LIN {X 0,Y 267.392,Z 674.93,A -85,B 0,C 180,E1 -18340.221,E2 -18340.221} C_VEL
LIN {X 0,Y 266.458,Z 688.326,A -85,B 0,C 180,E1 -18341.349,E2 -18341.349} C_VEL
LIN {X 0,Y 265.506,Z 700.294,A -85,B 0,C 180,E1 -18342.659,E2 -18342.659} C_VEL
LIN {X 0,Y 264.466,Z 712.728,A -85,B 0,C 180,E1 -18344.391,E2 -18344.391} C_VEL
LIN {X 0,Y 263.562,Z 722.705,A -85,B 0,C 180,E1 -18346.114,E2 -18346.114} C_VEL
LIN {X 0,Y 263.255,Z 725.943,A -85,B 0,C 180,E1 -18346.753,E2 -18346.753} C_VEL
LIN {X 0,Y 262.224,Z 730.137,A -85,B 0,C 180,E1 -18347.633,E2 -18347.633} C_VEL
LIN {X 0,Y 258.805,Z 736.401,A -85,B 0,C 180,E1 -18349.151,E2 -18349.151} C_VEL
LIN {X 0,Y 255.472,Z 742.099,A -85,B 0,C 180,E1 -18350.814,E2 -18350.814} C_VEL
LIN {X 0,Y 254.593,Z 745.41,A -85,B 0,C 180,E1 -18351.903,E2 -18351.903} C_VEL
LIN {X 0,Y 254.229,Z 751.934,A -85,B 0,C 180,E1 -18354.384,E2 -18354.384} C_VEL
LIN {X 0,Y 254.116,Z 756.958,A -85,B 0,C 180,E1 -18356.829,E2 -18356.829} C_VEL
LIN {X 0,Y 254.037,Z 760.636,A -85,B 0,C 180,E1 -18359.207,E2 -18359.207} C_VEL
LIN {X 0,Y 254.108,Z 763.255,A -85,B 0,C 180,E1 -18361.585,E2 -18361.585} C_VEL
LIN {X 0,Y 254.189,Z 764.422,A -85,B 0,C 180,E1 -18363.17,E2 -18363.17} C_VEL
LIN {X 0,Y 254.813,Z 765.536,A -85,B 0,C 180,E1 -18366.334,E2 -18366.334} C_VEL
LIN {X 0,Y 255.358,Z 765.437,A -85,B 0,C 180,E1 -18367.91,E2 -18367.91} C_VEL
LIN {X 0,Y 255.895,Z 764.932,A -85,B 0,C 180,E1 -18369.485,E2 -18369.485} C_VEL
LIN {X 0,Y 257.702,Z 762.72,A -85,B 0,C 180,E1 -18372.602,E2 -18372.602} C_VEL
LIN {X 0,Y 259.373,Z 759.949,A -85,B 0,C 180,E1 -18374.917,E2 -18374.917} C_VEL
LIN {X 0,Y 261.617,Z 756.12,A -85,B 0,C 180,E1 -18377.188,E2 -18377.188} C_VEL
LIN {X 0,Y 264.305,Z 751.227,A -85,B 0,C 180,E1 -18379.413,E2 -18379.413} C_VEL
LIN {X 0,Y 267.393,Z 745.066,A -85,B 0,C 180,E1 -18381.59,E2 -18381.59} C_VEL
LIN {X 0,Y 271.525,Z 736.165,A -85,B 0,C 180,E1 -18384.058,E2 -18384.058} C_VEL
LIN {X 0,Y 275.529,Z 726.618,A -85,B 0,C 180,E1 -18386.098,E2 -18386.098} C_VEL
LIN {X 0,Y 279.335,Z 716.352,A -85,B 0,C 180,E1 -18387.872,E2 -18387.872} C_VEL
LIN {X 0,Y 282.742,Z 706.311,A -85,B 0,C 180,E1 -18389.245,E2 -18389.245} C_VEL
LIN {X 0,Y 286.702,Z 692.836,A -85,B 0,C 180,E1 -18390.701,E2 -18390.701} C_VEL
LIN {X 0,Y 290.054,Z 679.318,A -85,B 0,C 180,E1 -18391.803,E2 -18391.803} C_VEL
LIN {X 0,Y 292.766,Z 665.226,A -85,B 0,C 180,E1 -18392.641,E2 -18392.641} C_VEL
LIN {X 0,Y 303.886,Z 598.397,A -85,B 0,C 180,E1 -18395.644,E2 -18395.644} C_VEL
LIN {X 0,Y 304.018,Z 586.794,A -85,B 0,C 180,E1 -18397.144,E2 -18397.144} C_VEL
LIN {X 0,Y 303.238,Z 583.136,A -85,B 0,C 180,E1 -18398.173,E2 -18398.173} C_VEL
LIN {X 0,Y 302.067,Z 579.008,A -85,B 0,C 180,E1 -18399.844,E2 -18399.844} C_VEL
LIN {X 0,Y 301.134,Z 575.43,A -85,B 0,C 180,E1 -18401.899,E2 -18401.899} C_VEL
LIN {X 0,Y 300.72,Z 573.5,A -85,B 0,C 180,E1 -18404.044,E2 -18404.044} C_VEL
LIN {X 0,Y 301.094,Z 572.833,A -85,B 0,C 180,E1 -18406.352,E2 -18406.352} C_VEL
LIN {X 0,Y 302.26,Z 573.558,A -85,B 0,C 180,E1 -18408.617,E2 -18408.617} C_VEL
LIN {X 0,Y 304.282,Z 575.713,A -85,B 0,C 180,E1 -18410.892,E2 -18410.892} C_VEL
LIN {X 0,Y 305.244,Z 577.018,A -85,B 0,C 180,E1 -18411.75,E2 -18411.75} C_VEL
LIN {X 0,Y 305.469,Z 578.807,A -85,B 0,C 180,E1 -18412.164,E2 -18412.164} C_VEL
LIN {X 0,Y 290.536,Z 664.644,A -85,B 0,C 180,E1 -18416.195,E2 -18416.195} C_VEL
LIN {X 0,Y 287.406,Z 682.317,A -85,B 0,C 180,E1 -18417.142,E2 -18417.142} C_VEL
LIN {X 0,Y 284.436,Z 695.44,A -85,B 0,C 180,E1 -18418.12,E2 -18418.12} C_VEL
LIN {X 0,Y 280.955,Z 708.177,A -85,B 0,C 180,E1 -18419.358,E2 -18419.358} C_VEL
LIN {X 0,Y 277.428,Z 719.855,A -85,B 0,C 180,E1 -18420.813,E2 -18420.813} C_VEL
LIN {X 0,Y 273.027,Z 732.546,A -85,B 0,C 180,E1 -18422.812,E2 -18422.812} C_VEL
LIN {X 0,Y 269.061,Z 742.824,A -85,B 0,C 180,E1 -18424.884,E2 -18424.884} C_VEL
LIN {X 0,Y 265.679,Z 751.358,A -85,B 0,C 180,E1 -18427.034,E2 -18427.034} C_VEL
LIN {X 0,Y 262.22,Z 759.42,A -85,B 0,C 180,E1 -18429.609,E2 -18429.609} C_VEL
LIN {X 0,Y 259.817,Z 765.006,A -85,B 0,C 180,E1 -18431.876,E2 -18431.876} C_VEL
LIN {X 0,Y 257.299,Z 770.761,A -85,B 0,C 180,E1 -18434.96,E2 -18434.96} C_VEL
LIN {X 0,Y 255.921,Z 773.892,A -85,B 0,C 180,E1 -18437.309,E2 -18437.309} C_VEL
LIN {X 0,Y 254.674,Z 776.576,A -85,B 0,C 180,E1 -18440.469,E2 -18440.469} C_VEL
LIN {X 0,Y 254.325,Z 777.326,A -85,B 0,C 180,E1 -18442.058,E2 -18442.058} C_VEL
LIN {X 0,Y 254.021,Z 777.636,A -85,B 0,C 180,E1 -18444.881,E2 -18444.881} C_VEL
LIN {X 0,Y 254.106,Z 777.04,A -85,B 0,C 180,E1 -18446.829,E2 -18446.829} C_VEL
LIN {X 0,Y 254.099,Z 775.415,A -85,B 0,C 180,E1 -18449.307,E2 -18449.307} C_VEL
LIN {X 0,Y 254.062,Z 777.171,A -85,B 0,C 180,E1 -18451.585,E2 -18451.585} C_VEL
LIN {X 0,Y 254.068,Z 777.92,A -85,B 0,C 180,E1 -18453.172,E2 -18453.172} C_VEL
LIN {X 0,Y 254.058,Z 778.293,A -85,B 0,C 180,E1 -18456.353,E2 -18456.353} C_VEL
LIN {X 0,Y 254.583,Z 777.255,A -85,B 0,C 180,E1 -18459.534,E2 -18459.534} C_VEL
LIN {X 0,Y 255.697,Z 774.838,A -85,B 0,C 180,E1 -18462.702,E2 -18462.702} C_VEL
LIN {X 0,Y 257.682,Z 771.008,A -85,B 0,C 180,E1 -18465.828,E2 -18465.828} C_VEL
LIN {X 0,Y 260.158,Z 765.718,A -85,B 0,C 180,E1 -18468.916,E2 -18468.916} C_VEL
LIN {X 0,Y 262.696,Z 760.659,A -85,B 0,C 180,E1 -18471.172,E2 -18471.172} C_VEL
LIN {X 0,Y 266.135,Z 753.523,A -85,B 0,C 180,E1 -18473.748,E2 -18473.748} C_VEL
LIN {X 0,Y 270.246,Z 744.85,A -85,B 0,C 180,E1 -18476.238,E2 -18476.238} C_VEL
LIN {X 0,Y 274.277,Z 735.941,A -85,B 0,C 180,E1 -18478.297,E2 -18478.297} C_VEL
LIN {X 0,Y 278.781,Z 725.251,A -85,B 0,C 180,E1 -18480.278,E2 -18480.278} C_VEL
LIN {X 0,Y 283.286,Z 713.812,A -85,B 0,C 180,E1 -18481.991,E2 -18481.991} C_VEL
LIN {X 0,Y 287.778,Z 700.836,A -85,B 0,C 180,E1 -18483.546,E2 -18483.546} C_VEL
LIN {X 0,Y 291.653,Z 688.544,A -85,B 0,C 180,E1 -18484.701,E2 -18484.701} C_VEL
LIN {X 0,Y 295.512,Z 674.017,A -85,B 0,C 180,E1 -18485.744,E2 -18485.744} C_VEL
LIN {X 0,Y 298.806,Z 658.507,A -85,B 0,C 180,E1 -18486.571,E2 -18486.571} C_VEL
LIN {X 0,Y 310.853,Z 589.993,A -85,B 0,C 180,E1 -18489.42,E2 -18489.42} C_VEL
LIN {X 0,Y 309.732,Z 587.337,A -85,B 0,C 180,E1 -18490.47,E2 -18490.47} C_VEL
LIN {X 0,Y 308.475,Z 584.65,A -85,B 0,C 180,E1 -18491.851,E2 -18491.851} C_VEL
LIN {X 0,Y 307.029,Z 581.664,A -85,B 0,C 180,E1 -18494.357,E2 -18494.357} C_VEL
LIN {X 0,Y 306.336,Z 581.501,A -85,B 0,C 180,E1 -18497.236,E2 -18497.236} C_VEL
LIN {X 0,Y 306.709,Z 582.69,A -85,B 0,C 180,E1 -18499.243,E2 -18499.243} C_VEL
LIN {X 0,Y 308.011,Z 587.255,A -85,B 0,C 180,E1 -18502.044,E2 -18502.044} C_VEL
LIN {X 0,Y 309.168,Z 591.574,A -85,B 0,C 180,E1 -18503.631,E2 -18503.631} C_VEL
LIN {X 0,Y 309.454,Z 593.023,A -85,B 0,C 180,E1 -18504.035,E2 -18504.035} C_VEL
LIN {X 0,Y 309.128,Z 598.033,A -85,B 0,C 180,E1 -18504.592,E2 -18504.592} C_VEL
LIN {X 0,Y 297.304,Z 660.919,A -85,B 0,C 180,E1 -18507.467,E2 -18507.467} C_VEL
LIN {X 0,Y 294.179,Z 674.017,A -85,B 0,C 180,E1 -18508.292,E2 -18508.292} C_VEL
LIN {X 0,Y 290.356,Z 687.818,A -85,B 0,C 180,E1 -18509.449,E2 -18509.449} C_VEL
LIN {X 0,Y 286.275,Z 700.375,A -85,B 0,C 180,E1 -18510.795,E2 -18510.795} C_VEL
LIN {X 0,Y 281.68,Z 712.899,A -85,B 0,C 180,E1 -18512.511,E2 -18512.511} C_VEL
LIN {X 0,Y 277.789,Z 722.415,A -85,B 0,C 180,E1 -18514.124,E2 -18514.124} C_VEL
LIN {X 0,Y 272.883,Z 733.435,A -85,B 0,C 180,E1 -18516.472,E2 -18516.472} C_VEL
LIN {X 0,Y 269.093,Z 741.153,A -85,B 0,C 180,E1 -18518.553,E2 -18518.553} C_VEL
LIN {X 0,Y 265.844,Z 747.53,A -85,B 0,C 180,E1 -18520.703,E2 -18520.703} C_VEL
LIN {X 0,Y 263.047,Z 752.715,A -85,B 0,C 180,E1 -18522.909,E2 -18522.909} C_VEL
LIN {X 0,Y 259.802,Z 758.061,A -85,B 0,C 180,E1 -18525.909,E2 -18525.909} C_VEL
LIN {X 0,Y 258.501,Z 760.04,A -85,B 0,C 180,E1 -18527.438,E2 -18527.438} C_VEL
LIN {X 0,Y 256.764,Z 762.528,A -85,B 0,C 180,E1 -18530.19,E2 -18530.19} C_VEL
LIN {X 0,Y 255.749,Z 763.559,A -85,B 0,C 180,E1 -18532.103,E2 -18532.103} C_VEL
LIN {X 0,Y 255.112,Z 763.932,A -85,B 0,C 180,E1 -18533.673,E2 -18533.673} C_VEL
LIN {X 0,Y 254.722,Z 763.876,A -85,B 0,C 180,E1 -18535.252,E2 -18535.252} C_VEL
LIN {X 0,Y 254.423,Z 763.427,A -85,B 0,C 180,E1 -18536.833,E2 -18536.833} C_VEL
LIN {X 0,Y 254.191,Z 762.579,A -85,B 0,C 180,E1 -18538.416,E2 -18538.416} C_VEL
LIN {X 0,Y 254.082,Z 761.32,A -85,B 0,C 180,E1 -18540,E2 -18540} C_VEL
LIN {X 0,Y 254.026,Z 758.577,A -85,B 0,C 180,E1 -18542.378,E2 -18542.378} C_VEL
LIN {X 0,Y 254.063,Z 754.795,A -85,B 0,C 180,E1 -18544.76,E2 -18544.76} C_VEL
LIN {X 0,Y 254.334,Z 749.877,A -85,B 0,C 180,E1 -18547.143,E2 -18547.143} C_VEL
LIN {X 0,Y 254.694,Z 743.632,A -85,B 0,C 180,E1 -18549.53,E2 -18549.53} C_VEL
LIN {X 0,Y 255.279,Z 735.844,A -85,B 0,C 180,E1 -18551.916,E2 -18551.916} C_VEL
LIN {X 0,Y 256.201,Z 726.268,A -85,B 0,C 180,E1 -18554.293,E2 -18554.293} C_VEL
LIN {X 0,Y 256.973,Z 716.914,A -85,B 0,C 180,E1 -18556.203,E2 -18556.203} C_VEL
LIN {X 0,Y 258.209,Z 705.975,A -85,B 0,C 180,E1 -18558.036,E2 -18558.036} C_VEL
LIN {X 0,Y 259.48,Z 693.061,A -85,B 0,C 180,E1 -18559.789,E2 -18559.789} C_VEL
LIN {X 0,Y 260.62,Z 679.32,A -85,B 0,C 180,E1 -18561.245,E2 -18561.245} C_VEL
LIN {X 0,Y 261.707,Z 665.038,A -85,B 0,C 180,E1 -18562.396,E2 -18562.396} C_VEL
LIN {X 0,Y 262.599,Z 649.769,A -85,B 0,C 180,E1 -18563.251,E2 -18563.251} C_VEL
LIN {X 0,Y 266.046,Z 579.424,A -85,B 0,C 180,E1 -18566.286,E2 -18566.286} C_VEL
LIN {X 0,Y 262.645,Z 547.859,A -85,B 0,C 180,E1 -18567.923,E2 -18567.923} C_VEL
LIN {X 0,Y 261.965,Z 538.359,A -85,B 0,C 180,E1 -18568.424,E2 -18568.424} C_VEL
LIN {X 0,Y 262.567,Z 533.905,A -85,B 0,C 180,E1 -18569.682,E2 -18569.682} C_VEL
LIN {X 0,Y 260.638,Z 524.372,A -85,B 0,C 180,E1 -18572.635,E2 -18572.635} C_VEL
LIN {X 0,Y 258.14,Z 512.652,A -85,B 0,C 180,E1 -18576.425,E2 -18576.425} C_VEL
LIN {X 0,Y 256.098,Z 503.706,A -85,B 0,C 180,E1 -18579.458,E2 -18579.458} C_VEL
LIN {X 0,Y 256.065,Z 503.713,A -85,B 0,C 180,E1 -18583.326,E2 -18583.326} C_VEL
LIN {X 0,Y 256.073,Z 503.714,A -85,B 0,C 180,E1 -18587.819,E2 -18587.819} C_VEL
LIN {X 0,Y 256.073,Z 503.711,A -85,B 0,C 180,E1 -18590.858,E2 -18590.858} C_VEL
LIN {X 0,Y 256.11,Z 503.704,A -85,B 0,C 180,E1 -18594.811,E2 -18594.811} C_VEL
LIN {X 0,Y 256.094,Z 503.707,A -85,B 0,C 180,E1 -18598.572,E2 -18598.572} C_VEL
LIN {X 0,Y 256.143,Z 503.701,A -85,B 0,C 180,E1 -18602.196,E2 -18602.196} C_VEL
LIN {X 0,Y 256.169,Z 503.701,A -85,B 0,C 180,E1 -18605.699,E2 -18605.699} C_VEL
LIN {X 0,Y 256.168,Z 503.7,A -85,B 0,C 180,E1 -18609.105,E2 -18609.105} C_VEL
LIN {X 0,Y 256.302,Z 503.682,A -85,B 0,C 180,E1 -18614.085,E2 -18614.085} C_VEL
LIN {X 0,Y 256.311,Z 503.681,A -85,B 0,C 180,E1 -18618.934,E2 -18618.934} C_VEL
LIN {X 0,Y 256.542,Z 503.651,A -85,B 0,C 180,E1 -18622.127,E2 -18622.127} C_VEL
LIN {X 0,Y 256.719,Z 503.628,A -85,B 0,C 180,E1 -18628.431,E2 -18628.431} C_VEL
LIN {X 0,Y 256.716,Z 503.633,A -85,B 0,C 180,E1 -18631.569,E2 -18631.569} C_VEL
LIN {X 0,Y 256.541,Z 503.651,A -85,B 0,C 180,E1 -18637.873,E2 -18637.873} C_VEL
LIN {X 0,Y 256.311,Z 503.682,A -85,B 0,C 180,E1 -18641.066,E2 -18641.066} C_VEL
LIN {X 0,Y 256.301,Z 503.681,A -85,B 0,C 180,E1 -18645.915,E2 -18645.915} C_VEL
LIN {X 0,Y 256.168,Z 503.699,A -85,B 0,C 180,E1 -18650.895,E2 -18650.895} C_VEL
LIN {X 0,Y 256.189,Z 503.697,A -85,B 0,C 180,E1 -18655.138,E2 -18655.138} C_VEL
LIN {X 0,Y 256.104,Z 503.709,A -85,B 0,C 180,E1 -18659.601,E2 -18659.601} C_VEL
LIN {X 0,Y 256.086,Z 503.711,A -85,B 0,C 180,E1 -18663.29,E2 -18663.29} C_VEL
LIN {X 0,Y 256.13,Z 503.707,A -85,B 0,C 180,E1 -18667.275,E2 -18667.275} C_VEL
LIN {X 0,Y 256.059,Z 503.715,A -85,B 0,C 180,E1 -18671.203,E2 -18671.203} C_VEL
LIN {X 0,Y 256.063,Z 503.714,A -85,B 0,C 180,E1 -18675.529,E2 -18675.529} C_VEL
LIN {X 0,Y 256.056,Z 503.713,A -85,B 0,C 180,E1 -18678.797,E2 -18678.797} C_VEL
LIN {X 0,Y 256.173,Z 503.781,A -85,B 0,C 180,E1 -18683.581,E2 -18683.581} C_VEL
LIN {X 0,Y 260.085,Z 520.834,A -85,B 0,C 180,E1 -18687.745,E2 -18687.745} C_VEL
LIN {X 0,Y 262.856,Z 533.76,A -85,B 0,C 180,E1 -18690.794,E2 -18690.794} C_VEL
LIN {X 0,Y 261.899,Z 545.387,A -85,B 0,C 180,E1 -18693.29,E2 -18693.29} C_VEL
LIN {X 0,Y 261.425,Z 550.677,A -85,B 0,C 180,E1 -18694.364,E2 -18694.364} C_VEL
LIN {X 0,Y 263.474,Z 573.72,A -85,B 0,C 180,E1 -18695.465,E2 -18695.465} C_VEL
LIN {X 0,Y 264.373,Z 582.285,A -85,B 0,C 180,E1 -18695.876,E2 -18695.876} C_VEL
LIN {X 0,Y 261.074,Z 660.539,A -85,B 0,C 180,E1 -18699.206,E2 -18699.206} C_VEL
LIN {X 0,Y 260.346,Z 674.677,A -85,B 0,C 180,E1 -18700.074,E2 -18700.074} C_VEL
LIN {X 0,Y 259.423,Z 687.6,A -85,B 0,C 180,E1 -18701.182,E2 -18701.182} C_VEL
LIN {X 0,Y 258.394,Z 700.276,A -85,B 0,C 180,E1 -18702.591,E2 -18702.591} C_VEL
LIN {X 0,Y 257.367,Z 712.658,A -85,B 0,C 180,E1 -18704.356,E2 -18704.356} C_VEL
LIN {X 0,Y 256.452,Z 722.704,A -85,B 0,C 180,E1 -18706.126,E2 -18706.126} C_VEL
LIN {X 0,Y 255.507,Z 733.568,A -85,B 0,C 180,E1 -18708.497,E2 -18708.497} C_VEL
LIN {X 0,Y 254.813,Z 742.226,A -85,B 0,C 180,E1 -18710.875,E2 -18710.875} C_VEL
LIN {X 0,Y 254.593,Z 745.41,A -85,B 0,C 180,E1 -18711.903,E2 -18711.903} C_VEL
LIN {X 0,Y 253.763,Z 748.506,A -85,B 0,C 180,E1 -18713.022,E2 -18713.022} C_VEL
LIN {X 0,Y 250.712,Z 752.886,A -85,B 0,C 180,E1 -18714.919,E2 -18714.919} C_VEL
LIN {X 0,Y 247.72,Z 756.704,A -85,B 0,C 180,E1 -18716.932,E2 -18716.932} C_VEL
LIN {X 0,Y 247.008,Z 758.795,A -85,B 0,C 180,E1 -18718.21,E2 -18718.21} C_VEL
LIN {X 0,Y 246.984,Z 761.253,A -85,B 0,C 180,E1 -18720,E2 -18720} C_VEL
LIN {X 0,Y 247.04,Z 763.011,A -85,B 0,C 180,E1 -18721.63,E2 -18721.63} C_VEL
LIN {X 0,Y 247.113,Z 764.353,A -85,B 0,C 180,E1 -18723.261,E2 -18723.261} C_VEL
LIN {X 0,Y 247.336,Z 765.232,A -85,B 0,C 180,E1 -18724.89,E2 -18724.89} C_VEL
LIN {X 0,Y 248.143,Z 765.789,A -85,B 0,C 180,E1 -18727.57,E2 -18727.57} C_VEL
LIN {X 0,Y 248.911,Z 765.442,A -85,B 0,C 180,E1 -18729.754,E2 -18729.754} C_VEL
LIN {X 0,Y 249.753,Z 764.668,A -85,B 0,C 180,E1 -18731.36,E2 -18731.36} C_VEL
LIN {X 0,Y 250.832,Z 763.486,A -85,B 0,C 180,E1 -18732.953,E2 -18732.953} C_VEL
LIN {X 0,Y 253.27,Z 759.929,A -85,B 0,C 180,E1 -18736.111,E2 -18736.111} C_VEL
LIN {X 0,Y 255.871,Z 756.046,A -85,B 0,C 180,E1 -18738.413,E2 -18738.413} C_VEL
LIN {X 0,Y 258.819,Z 751.037,A -85,B 0,C 180,E1 -18740.671,E2 -18740.671} C_VEL
LIN {X 0,Y 262.845,Z 743.72,A -85,B 0,C 180,E1 -18743.228,E2 -18743.228} C_VEL
LIN {X 0,Y 266.715,Z 735.856,A -85,B 0,C 180,E1 -18745.353,E2 -18745.353} C_VEL
LIN {X 0,Y 271.072,Z 726.284,A -85,B 0,C 180,E1 -18747.4,E2 -18747.4} C_VEL
LIN {X 0,Y 274.86,Z 716.69,A -85,B 0,C 180,E1 -18749.066,E2 -18749.066} C_VEL
LIN {X 0,Y 278.843,Z 705.849,A -85,B 0,C 180,E1 -18750.545,E2 -18750.545} C_VEL
LIN {X 0,Y 282.722,Z 693.433,A -85,B 0,C 180,E1 -18751.887,E2 -18751.887} C_VEL
LIN {X 0,Y 286.314,Z 680.01,A -85,B 0,C 180,E1 -18752.999,E2 -18752.999} C_VEL
LIN {X 0,Y 289.331,Z 665.633,A -85,B 0,C 180,E1 -18753.86,E2 -18753.86} C_VEL
LIN {X 0,Y 300.893,Z 600.866,A -85,B 0,C 180,E1 -18756.784,E2 -18756.784} C_VEL
LIN {X 0,Y 301.233,Z 591.187,A -85,B 0,C 180,E1 -18758.088,E2 -18758.088} C_VEL
LIN {X 0,Y 300.317,Z 586.941,A -85,B 0,C 180,E1 -18759.567,E2 -18759.567} C_VEL
LIN {X 0,Y 299.382,Z 582.854,A -85,B 0,C 180,E1 -18761.663,E2 -18761.663} C_VEL
LIN {X 0,Y 299.013,Z 581.024,A -85,B 0,C 180,E1 -18763.229,E2 -18763.229} C_VEL
LIN {X 0,Y 299.006,Z 579.899,A -85,B 0,C 180,E1 -18765.159,E2 -18765.159} C_VEL
LIN {X 0,Y 299.624,Z 579.8,A -85,B 0,C 180,E1 -18767.138,E2 -18767.138} C_VEL
LIN {X 0,Y 300.971,Z 580.983,A -85,B 0,C 180,E1 -18769.288,E2 -18769.288} C_VEL
LIN {X 0,Y 302.623,Z 582.886,A -85,B 0,C 180,E1 -18771.054,E2 -18771.054} C_VEL
LIN {X 0,Y 286.983,Z 666.845,A -85,B 0,C 180,E1 -18775.026,E2 -18775.026} C_VEL
LIN {X 0,Y 284.073,Z 681.963,A -85,B 0,C 180,E1 -18775.855,E2 -18775.855} C_VEL
LIN {X 0,Y 280.837,Z 694.936,A -85,B 0,C 180,E1 -18776.809,E2 -18776.809} C_VEL
LIN {X 0,Y 276.708,Z 708.994,A -85,B 0,C 180,E1 -18778.195,E2 -18778.195} C_VEL
LIN {X 0,Y 272.872,Z 720.308,A -85,B 0,C 180,E1 -18779.638,E2 -18779.638} C_VEL
LIN {X 0,Y 268.584,Z 731.799,A -85,B 0,C 180,E1 -18781.475,E2 -18781.475} C_VEL
LIN {X 0,Y 264.27,Z 742.093,A -85,B 0,C 180,E1 -18783.548,E2 -18783.548} C_VEL
LIN {X 0,Y 260.479,Z 750.625,A -85,B 0,C 180,E1 -18785.703,E2 -18785.703} C_VEL
LIN {X 0,Y 256.677,Z 758.745,A -85,B 0,C 180,E1 -18788.307,E2 -18788.307} C_VEL
LIN {X 0,Y 253.947,Z 764.349,A -85,B 0,C 180,E1 -18790.604,E2 -18790.604} C_VEL
LIN {X 0,Y 251.722,Z 768.883,A -85,B 0,C 180,E1 -18792.953,E2 -18792.953} C_VEL
LIN {X 0,Y 249.877,Z 772.4,A -85,B 0,C 180,E1 -18795.337,E2 -18795.337} C_VEL
LIN {X 0,Y 248.214,Z 775.619,A -85,B 0,C 180,E1 -18798.568,E2 -18798.568} C_VEL
LIN {X 0,Y 247.649,Z 776.637,A -85,B 0,C 180,E1 -18800.196,E2 -18800.196} C_VEL
LIN {X 0,Y 247.273,Z 777.224,A -85,B 0,C 180,E1 -18801.83,E2 -18801.83} C_VEL
LIN {X 0,Y 246.944,Z 777.216,A -85,B 0,C 180,E1 -18804.937,E2 -18804.937} C_VEL
LIN {X 0,Y 247.037,Z 776.558,A -85,B 0,C 180,E1 -18806.738,E2 -18806.738} C_VEL
LIN {X 0,Y 247.028,Z 774.794,A -85,B 0,C 180,E1 -18809.389,E2 -18809.389} C_VEL
LIN {X 0,Y 246.993,Z 776.557,A -85,B 0,C 180,E1 -18811.631,E2 -18811.631} C_VEL
LIN {X 0,Y 247.003,Z 777.411,A -85,B 0,C 180,E1 -18813.262,E2 -18813.262} C_VEL
LIN {X 0,Y 247.001,Z 778.015,A -85,B 0,C 180,E1 -18816.535,E2 -18816.535} C_VEL
LIN {X 0,Y 247.563,Z 777.226,A -85,B 0,C 180,E1 -18819.807,E2 -18819.807} C_VEL
LIN {X 0,Y 248.742,Z 775.065,A -85,B 0,C 180,E1 -18823.064,E2 -18823.064} C_VEL
LIN {X 0,Y 250.844,Z 771.492,A -85,B 0,C 180,E1 -18826.271,E2 -18826.271} C_VEL
LIN {X 0,Y 253.501,Z 766.481,A -85,B 0,C 180,E1 -18829.432,E2 -18829.432} C_VEL
LIN {X 0,Y 257.057,Z 759.913,A -85,B 0,C 180,E1 -18832.505,E2 -18832.505} C_VEL
LIN {X 0,Y 261.536,Z 751.621,A -85,B 0,C 180,E1 -18835.465,E2 -18835.465} C_VEL
LIN {X 0,Y 266.126,Z 742.578,A -85,B 0,C 180,E1 -18837.954,E2 -18837.954} C_VEL
LIN {X 0,Y 270.579,Z 733.388,A -85,B 0,C 180,E1 -18840,E2 -18840} C_VEL
LIN {X 0,Y 275.519,Z 722.392,A -85,B 0,C 180,E1 -18841.958,E2 -18841.958} C_VEL
LIN {X 0,Y 280.898,Z 709.192,A -85,B 0,C 180,E1 -18843.827,E2 -18843.827} C_VEL
LIN {X 0,Y 285.737,Z 695.665,A -85,B 0,C 180,E1 -18845.311,E2 -18845.311} C_VEL
LIN {X 0,Y 289.969,Z 682.313,A -85,B 0,C 180,E1 -18846.428,E2 -18846.428} C_VEL
LIN {X 0,Y 293.827,Z 667.571,A -85,B 0,C 180,E1 -18847.369,E2 -18847.369} C_VEL
LIN {X 0,Y 297.165,Z 650.661,A -85,B 0,C 180,E1 -18848.169,E2 -18848.169} C_VEL
LIN {X 0,Y 307.759,Z 594.745,A -85,B 0,C 180,E1 -18850.483,E2 -18850.483} C_VEL
LIN {X 0,Y 307.584,Z 593.986,A -85,B 0,C 180,E1 -18850.736,E2 -18850.736} C_VEL
LIN {X 0,Y 306.397,Z 591.182,A -85,B 0,C 180,E1 -18852.197,E2 -18852.197} C_VEL
LIN {X 0,Y 305.201,Z 588.506,A -85,B 0,C 180,E1 -18854.451,E2 -18854.451} C_VEL
LIN {X 0,Y 304.623,Z 588.275,A -85,B 0,C 180,E1 -18856.201,E2 -18856.201} C_VEL
LIN {X 0,Y 304.654,Z 588.85,A -85,B 0,C 180,E1 -18858.315,E2 -18858.315} C_VEL
LIN {X 0,Y 304.836,Z 589.737,A -85,B 0,C 180,E1 -18859.221,E2 -18859.221} C_VEL
LIN {X 0,Y 305.833,Z 593.701,A -85,B 0,C 180,E1 -18861.65,E2 -18861.65} C_VEL
LIN {X 0,Y 306.676,Z 597.433,A -85,B 0,C 180,E1 -18863.053,E2 -18863.053} C_VEL
LIN {X 0,Y 306.59,Z 599.523,A -85,B 0,C 180,E1 -18863.376,E2 -18863.376} C_VEL
LIN {X 0,Y 294.42,Z 660.456,A -85,B 0,C 180,E1 -18866.187,E2 -18866.187} C_VEL
LIN {X 0,Y 290.88,Z 674.642,A -85,B 0,C 180,E1 -18867.069,E2 -18867.069} C_VEL
LIN {X 0,Y 287.312,Z 686.628,A -85,B 0,C 180,E1 -18868.064,E2 -18868.064} C_VEL
LIN {X 0,Y 282.881,Z 699.295,A -85,B 0,C 180,E1 -18869.382,E2 -18869.382} C_VEL
LIN {X 0,Y 278.462,Z 710.921,A -85,B 0,C 180,E1 -18870.932,E2 -18870.932} C_VEL
LIN {X 0,Y 273.425,Z 722.406,A -85,B 0,C 180,E1 -18872.855,E2 -18872.855} C_VEL
LIN {X 0,Y 268.9,Z 731.998,A -85,B 0,C 180,E1 -18874.868,E2 -18874.868} C_VEL
LIN {X 0,Y 264.681,Z 739.954,A -85,B 0,C 180,E1 -18876.943,E2 -18876.943} C_VEL
LIN {X 0,Y 261.607,Z 745.554,A -85,B 0,C 180,E1 -18878.735,E2 -18878.735} C_VEL
LIN {X 0,Y 258.361,Z 751.101,A -85,B 0,C 180,E1 -18880.948,E2 -18880.948} C_VEL
LIN {X 0,Y 255.531,Z 755.641,A -85,B 0,C 180,E1 -18883.215,E2 -18883.215} C_VEL
LIN {X 0,Y 253.019,Z 759.166,A -85,B 0,C 180,E1 -18885.523,E2 -18885.523} C_VEL
LIN {X 0,Y 251.647,Z 760.99,A -85,B 0,C 180,E1 -18887.09,E2 -18887.09} C_VEL
LIN {X 0,Y 249.704,Z 763.336,A -85,B 0,C 180,E1 -18890.094,E2 -18890.094} C_VEL
LIN {X 0,Y 248.749,Z 764.025,A -85,B 0,C 180,E1 -18891.879,E2 -18891.879} C_VEL
LIN {X 0,Y 248.061,Z 764.243,A -85,B 0,C 180,E1 -18893.493,E2 -18893.493} C_VEL
LIN {X 0,Y 247.658,Z 764.067,A -85,B 0,C 180,E1 -18895.116,E2 -18895.116} C_VEL
LIN {X 0,Y 247.341,Z 763.497,A -85,B 0,C 180,E1 -18896.742,E2 -18896.742} C_VEL
LIN {X 0,Y 247.122,Z 762.51,A -85,B 0,C 180,E1 -18898.37,E2 -18898.37} C_VEL
LIN {X 0,Y 247.011,Z 761.087,A -85,B 0,C 180,E1 -18900,E2 -18900} C_VEL
LIN {X 0,Y 246.944,Z 758.157,A -85,B 0,C 180,E1 -18902.447,E2 -18902.447} C_VEL
LIN {X 0,Y 247.028,Z 753.408,A -85,B 0,C 180,E1 -18905.275,E2 -18905.275} C_VEL
LIN {X 0,Y 247.37,Z 746.952,A -85,B 0,C 180,E1 -18908.167,E2 -18908.167} C_VEL
LIN {X 0,Y 247.841,Z 739.956,A -85,B 0,C 180,E1 -18910.621,E2 -18910.621} C_VEL
LIN {X 0,Y 248.604,Z 731.318,A -85,B 0,C 180,E1 -18913.071,E2 -18913.071} C_VEL
LIN {X 0,Y 249.447,Z 722.549,A -85,B 0,C 180,E1 -18915.106,E2 -18915.106} C_VEL
LIN {X 0,Y 250.454,Z 712.115,A -85,B 0,C 180,E1 -18917.115,E2 -18917.115} C_VEL
LIN {X 0,Y 251.657,Z 700.391,A -85,B 0,C 180,E1 -18918.944,E2 -18918.944} C_VEL
LIN {X 0,Y 252.912,Z 687.767,A -85,B 0,C 180,E1 -18920.538,E2 -18920.538} C_VEL
LIN {X 0,Y 254.056,Z 673.522,A -85,B 0,C 180,E1 -18921.929,E2 -18921.929} C_VEL
LIN {X 0,Y 255.01,Z 659.339,A -85,B 0,C 180,E1 -18922.963,E2 -18922.963} C_VEL
LIN {X 0,Y 256.145,Z 638.79,A -85,B 0,C 180,E1 -18923.98,E2 -18923.98} C_VEL
LIN {X 0,Y 259.188,Z 580.447,A -85,B 0,C 180,E1 -18926.608,E2 -18926.608} C_VEL
LIN {X 0,Y 255.807,Z 548.384,A -85,B 0,C 180,E1 -18928.315,E2 -18928.315} C_VEL
LIN {X 0,Y 255.078,Z 538.33,A -85,B 0,C 180,E1 -18928.843,E2 -18928.843} C_VEL
LIN {X 0,Y 255.532,Z 535.448,A -85,B 0,C 180,E1 -18929.674,E2 -18929.674} C_VEL
LIN {X 0,Y 254.41,Z 529.1,A -85,B 0,C 180,E1 -18931.659,E2 -18931.659} C_VEL
LIN {X 0,Y 252.025,Z 517.77,A -85,B 0,C 180,E1 -18935.355,E2 -18935.355} C_VEL
LIN {X 0,Y 249.457,Z 506.488,A -85,B 0,C 180,E1 -18939.216,E2 -18939.216} C_VEL
LIN {X 0,Y 249.027,Z 504.587,A -85,B 0,C 180,E1 -18939.932,E2 -18939.932} C_VEL
LIN {X 0,Y 249.014,Z 504.589,A -85,B 0,C 180,E1 -18942.793,E2 -18942.793} C_VEL
LIN {X 0,Y 249.017,Z 504.593,A -85,B 0,C 180,E1 -18947.363,E2 -18947.363} C_VEL
LIN {X 0,Y 249.045,Z 504.586,A -85,B 0,C 180,E1 -18952.2,E2 -18952.2} C_VEL
LIN {X 0,Y 249.058,Z 504.586,A -85,B 0,C 180,E1 -18955.641,E2 -18955.641} C_VEL
LIN {X 0,Y 249.054,Z 504.588,A -85,B 0,C 180,E1 -18959.473,E2 -18959.473} C_VEL
LIN {X 0,Y 249.075,Z 504.583,A -85,B 0,C 180,E1 -18963.162,E2 -18963.162} C_VEL
LIN {X 0,Y 249.081,Z 504.581,A -85,B 0,C 180,E1 -18966.733,E2 -18966.733} C_VEL
LIN {X 0,Y 249.112,Z 504.577,A -85,B 0,C 180,E1 -18970.211,E2 -18970.211} C_VEL
LIN {X 0,Y 249.243,Z 504.564,A -85,B 0,C 180,E1 -18973.622,E2 -18973.622} C_VEL
LIN {X 0,Y 249.254,Z 504.559,A -85,B 0,C 180,E1 -18978.616,E2 -18978.616} C_VEL
LIN {X 0,Y 249.486,Z 504.531,A -85,B 0,C 180,E1 -18981.903,E2 -18981.903} C_VEL
LIN {X 0,Y 249.443,Z 504.536,A -85,B 0,C 180,E1 -18986.77,E2 -18986.77} C_VEL
LIN {X 0,Y 249.737,Z 504.498,A -85,B 0,C 180,E1 -18990,E2 -18990} C_VEL
LIN {X 0,Y 249.439,Z 504.539,A -85,B 0,C 180,E1 -18993.23,E2 -18993.23} C_VEL
LIN {X 0,Y 249.485,Z 504.529,A -85,B 0,C 180,E1 -18998.097,E2 -18998.097} C_VEL
LIN {X 0,Y 249.254,Z 504.563,A -85,B 0,C 180,E1 -19001.383,E2 -19001.383} C_VEL
LIN {X 0,Y 249.243,Z 504.559,A -85,B 0,C 180,E1 -19006.378,E2 -19006.378} C_VEL
LIN {X 0,Y 249.088,Z 504.583,A -85,B 0,C 180,E1 -19011.518,E2 -19011.518} C_VEL
LIN {X 0,Y 249.131,Z 504.577,A -85,B 0,C 180,E1 -19015.482,E2 -19015.482} C_VEL
LIN {X 0,Y 249.074,Z 504.584,A -85,B 0,C 180,E1 -19018.989,E2 -19018.989} C_VEL
LIN {X 0,Y 249.037,Z 504.585,A -85,B 0,C 180,E1 -19022.425,E2 -19022.425} C_VEL
LIN {X 0,Y 249.07,Z 504.582,A -85,B 0,C 180,E1 -19026.339,E2 -19026.339} C_VEL
LIN {X 0,Y 249.027,Z 504.587,A -85,B 0,C 180,E1 -19030.474,E2 -19030.474} C_VEL
LIN {X 0,Y 249.008,Z 504.591,A -85,B 0,C 180,E1 -19034.878,E2 -19034.878} C_VEL
LIN {X 0,Y 249.019,Z 504.592,A -85,B 0,C 180,E1 -19037.363,E2 -19037.363} C_VEL
LIN {X 0,Y 249.045,Z 504.587,A -85,B 0,C 180,E1 -19042.2,E2 -19042.2} C_VEL
LIN {X 0,Y 249.111,Z 504.704,A -85,B 0,C 180,E1 -19043.201,E2 -19043.201} C_VEL
LIN {X 0,Y 253.095,Z 522.045,A -85,B 0,C 180,E1 -19047.519,E2 -19047.519} C_VEL
LIN {X 0,Y 255.642,Z 533.748,A -85,B 0,C 180,E1 -19050.34,E2 -19050.34} C_VEL
LIN {X 0,Y 255.822,Z 537.179,A -85,B 0,C 180,E1 -19051.122,E2 -19051.122} C_VEL
LIN {X 0,Y 254.468,Z 550.592,A -85,B 0,C 180,E1 -19054.012,E2 -19054.012} C_VEL
LIN {X 0,Y 256.447,Z 573.918,A -85,B 0,C 180,E1 -19055.171,E2 -19055.171} C_VEL
LIN {X 0,Y 257.365,Z 583.014,A -85,B 0,C 180,E1 -19055.622,E2 -19055.622} C_VEL
LIN {X 0,Y 253.994,Z 660.979,A -85,B 0,C 180,E1 -19059.077,E2 -19059.077} C_VEL
LIN {X 0,Y 253.211,Z 675.633,A -85,B 0,C 180,E1 -19060.017,E2 -19060.017} C_VEL
LIN {X 0,Y 252.219,Z 690.104,A -85,B 0,C 180,E1 -19061.334,E2 -19061.334} C_VEL
LIN {X 0,Y 250.996,Z 703.105,A -85,B 0,C 180,E1 -19062.902,E2 -19062.902} C_VEL
LIN {X 0,Y 250.269,Z 712.589,A -85,B 0,C 180,E1 -19064.319,E2 -19064.319} C_VEL
LIN {X 0,Y 249.356,Z 722.664,A -85,B 0,C 180,E1 -19066.139,E2 -19066.139} C_VEL
LIN {X 0,Y 248.384,Z 733.499,A -85,B 0,C 180,E1 -19068.576,E2 -19068.576} C_VEL
LIN {X 0,Y 247.713,Z 742.177,A -85,B 0,C 180,E1 -19071.023,E2 -19071.023} C_VEL
LIN {X 0,Y 247.319,Z 749.172,A -85,B 0,C 180,E1 -19073.473,E2 -19073.473} C_VEL
LIN {X 0,Y 247.075,Z 754.745,A -85,B 0,C 180,E1 -19075.922,E2 -19075.922} C_VEL
LIN {X 0,Y 247.008,Z 758.795,A -85,B 0,C 180,E1 -19078.21,E2 -19078.21} C_VEL
LIN {X 0,Y 246.298,Z 760.705,A -85,B 0,C 180,E1 -19079.498,E2 -19079.498} C_VEL
LIN {X 0,Y 243.425,Z 763.108,A -85,B 0,C 180,E1 -19081.65,E2 -19081.65} C_VEL
LIN {X 0,Y 241.128,Z 764.436,A -85,B 0,C 180,E1 -19083.436,E2 -19083.436} C_VEL
LIN {X 0,Y 240.308,Z 765.15,A -85,B 0,C 180,E1 -19084.831,E2 -19084.831} C_VEL
LIN {X 0,Y 240.328,Z 765.338,A -85,B 0,C 180,E1 -19085.302,E2 -19085.302} C_VEL
LIN {X 0,Y 240.934,Z 765.973,A -85,B 0,C 180,E1 -19087.352,E2 -19087.352} C_VEL
LIN {X 0,Y 241.921,Z 765.862,A -85,B 0,C 180,E1 -19090.038,E2 -19090.038} C_VEL
LIN {X 0,Y 242.817,Z 765.269,A -85,B 0,C 180,E1 -19091.689,E2 -19091.689} C_VEL
LIN {X 0,Y 243.953,Z 764.267,A -85,B 0,C 180,E1 -19093.325,E2 -19093.325} C_VEL
LIN {X 0,Y 246.544,Z 761.032,A -85,B 0,C 180,E1 -19096.563,E2 -19096.563} C_VEL
LIN {X 0,Y 249.286,Z 757.426,A -85,B 0,C 180,E1 -19098.918,E2 -19098.918} C_VEL
LIN {X 0,Y 252.389,Z 752.812,A -85,B 0,C 180,E1 -19101.223,E2 -19101.223} C_VEL
LIN {X 0,Y 255.972,Z 746.981,A -85,B 0,C 180,E1 -19103.46,E2 -19103.46} C_VEL
LIN {X 0,Y 259.965,Z 739.902,A -85,B 0,C 180,E1 -19105.63,E2 -19105.63} C_VEL
LIN {X 0,Y 264.388,Z 731.179,A -85,B 0,C 180,E1 -19107.722,E2 -19107.722} C_VEL
LIN {X 0,Y 269.167,Z 720.687,A -85,B 0,C 180,E1 -19109.742,E2 -19109.742} C_VEL
LIN {X 0,Y 274.028,Z 708.704,A -85,B 0,C 180,E1 -19111.504,E2 -19111.504} C_VEL
LIN {X 0,Y 278.249,Z 696.588,A -85,B 0,C 180,E1 -19112.891,E2 -19112.891} C_VEL
LIN {X 0,Y 282.245,Z 683.046,A -85,B 0,C 180,E1 -19114.074,E2 -19114.074} C_VEL
LIN {X 0,Y 285.551,Z 669.324,A -85,B 0,C 180,E1 -19114.96,E2 -19114.96} C_VEL
LIN {X 0,Y 298.195,Z 603.054,A -85,B 0,C 180,E1 -19118.003,E2 -19118.003} C_VEL
LIN {X 0,Y 298.617,Z 596.109,A -85,B 0,C 180,E1 -19118.984,E2 -19118.984} C_VEL
LIN {X 0,Y 297.827,Z 591.829,A -85,B 0,C 180,E1 -19120.673,E2 -19120.673} C_VEL
LIN {X 0,Y 297.328,Z 588.63,A -85,B 0,C 180,E1 -19122.56,E2 -19122.56} C_VEL
LIN {X 0,Y 297.184,Z 587.035,A -85,B 0,C 180,E1 -19124.592,E2 -19124.592} C_VEL
LIN {X 0,Y 297.788,Z 586.633,A -85,B 0,C 180,E1 -19127.023,E2 -19127.023} C_VEL
LIN {X 0,Y 299.152,Z 587.847,A -85,B 0,C 180,E1 -19129.258,E2 -19129.258} C_VEL
LIN {X 0,Y 299.704,Z 588.601,A -85,B 0,C 180,E1 -19129.978,E2 -19129.978} C_VEL
LIN {X 0,Y 283.772,Z 669.022,A -85,B 0,C 180,E1 -19133.806,E2 -19133.806} C_VEL
LIN {X 0,Y 280.424,Z 684.304,A -85,B 0,C 180,E1 -19134.69,E2 -19134.69} C_VEL
LIN {X 0,Y 276.518,Z 698.155,A -85,B 0,C 180,E1 -19135.783,E2 -19135.783} C_VEL
LIN {X 0,Y 272.61,Z 710.09,A -85,B 0,C 180,E1 -19137.002,E2 -19137.002} C_VEL
LIN {X 0,Y 267.697,Z 723.242,A -85,B 0,C 180,E1 -19138.768,E2 -19138.768} C_VEL
LIN {X 0,Y 262.719,Z 734.903,A -85,B 0,C 180,E1 -19140.777,E2 -19140.777} C_VEL
LIN {X 0,Y 258.223,Z 744.587,A -85,B 0,C 180,E1 -19142.878,E2 -19142.878} C_VEL
LIN {X 0,Y 253.631,Z 753.744,A -85,B 0,C 180,E1 -19145.44,E2 -19145.44} C_VEL
LIN {X 0,Y 250.226,Z 760.176,A -85,B 0,C 180,E1 -19147.718,E2 -19147.718} C_VEL
LIN {X 0,Y 247.345,Z 765.446,A -85,B 0,C 180,E1 -19150.064,E2 -19150.064} C_VEL
LIN {X 0,Y 244.981,Z 769.637,A -85,B 0,C 180,E1 -19152.469,E2 -19152.469} C_VEL
LIN {X 0,Y 243.015,Z 772.879,A -85,B 0,C 180,E1 -19154.913,E2 -19154.913} C_VEL
LIN {X 0,Y 242.035,Z 774.541,A -85,B 0,C 180,E1 -19156.568,E2 -19156.568} C_VEL
LIN {X 0,Y 240.639,Z 776.609,A -85,B 0,C 180,E1 -19159.908,E2 -19159.908} C_VEL
LIN {X 0,Y 239.959,Z 777.123,A -85,B 0,C 180,E1 -19163.272,E2 -19163.272} C_VEL
LIN {X 0,Y 239.881,Z 776.766,A -85,B 0,C 180,E1 -19164.958,E2 -19164.958} C_VEL
LIN {X 0,Y 239.968,Z 775.97,A -85,B 0,C 180,E1 -19166.642,E2 -19166.642} C_VEL
LIN {X 0,Y 239.987,Z 773.975,A -85,B 0,C 180,E1 -19169.371,E2 -19169.371} C_VEL
LIN {X 0,Y 239.925,Z 775.926,A -85,B 0,C 180,E1 -19171.679,E2 -19171.679} C_VEL
LIN {X 0,Y 239.938,Z 776.882,A -85,B 0,C 180,E1 -19173.359,E2 -19173.359} C_VEL
LIN {X 0,Y 239.941,Z 777.696,A -85,B 0,C 180,E1 -19176.728,E2 -19176.728} C_VEL
LIN {X 0,Y 240.528,Z 777.131,A -85,B 0,C 180,E1 -19180.097,E2 -19180.097} C_VEL
LIN {X 0,Y 241.797,Z 775.217,A -85,B 0,C 180,E1 -19183.446,E2 -19183.446} C_VEL
LIN {X 0,Y 244.031,Z 771.943,A -85,B 0,C 180,E1 -19186.738,E2 -19186.738} C_VEL
LIN {X 0,Y 246.866,Z 767.275,A -85,B 0,C 180,E1 -19189.976,E2 -19189.976} C_VEL
LIN {X 0,Y 250.613,Z 761.082,A -85,B 0,C 180,E1 -19193.117,E2 -19193.117} C_VEL
LIN {X 0,Y 254.662,Z 754.259,A -85,B 0,C 180,E1 -19195.764,E2 -19195.764} C_VEL
LIN {X 0,Y 260.112,Z 744.667,A -85,B 0,C 180,E1 -19198.659,E2 -19198.659} C_VEL
LIN {X 0,Y 264.719,Z 735.936,A -85,B 0,C 180,E1 -19200.735,E2 -19200.735} C_VEL
LIN {X 0,Y 269.888,Z 725.656,A -85,B 0,C 180,E1 -19202.707,E2 -19202.707} C_VEL
LIN {X 0,Y 274.972,Z 714.364,A -85,B 0,C 180,E1 -19204.437,E2 -19204.437} C_VEL
LIN {X 0,Y 280.435,Z 700.926,A -85,B 0,C 180,E1 -19206.082,E2 -19206.082} C_VEL
LIN {X 0,Y 284.795,Z 688.87,A -85,B 0,C 180,E1 -19207.2,E2 -19207.2} C_VEL
LIN {X 0,Y 289.557,Z 673.058,A -85,B 0,C 180,E1 -19208.349,E2 -19208.349} C_VEL
LIN {X 0,Y 293.238,Z 657.818,A -85,B 0,C 180,E1 -19209.152,E2 -19209.152} C_VEL
LIN {X 0,Y 304.926,Z 599.413,A -85,B 0,C 180,E1 -19211.597,E2 -19211.597} C_VEL
LIN {X 0,Y 304.185,Z 597.426,A -85,B 0,C 180,E1 -19212.744,E2 -19212.744} C_VEL
LIN {X 0,Y 303.253,Z 595.304,A -85,B 0,C 180,E1 -19214.73,E2 -19214.73} C_VEL
LIN {X 0,Y 302.724,Z 595.182,A -85,B 0,C 180,E1 -19216.74,E2 -19216.74} C_VEL
LIN {X 0,Y 302.848,Z 595.851,A -85,B 0,C 180,E1 -19218.503,E2 -19218.503} C_VEL
LIN {X 0,Y 303.619,Z 599.848,A -85,B 0,C 180,E1 -19221.136,E2 -19221.136} C_VEL
LIN {X 0,Y 304.07,Z 602.499,A -85,B 0,C 180,E1 -19222.206,E2 -19222.206} C_VEL
LIN {X 0,Y 291.464,Z 662.003,A -85,B 0,C 180,E1 -19224.957,E2 -19224.957} C_VEL
LIN {X 0,Y 287.768,Z 675.658,A -85,B 0,C 180,E1 -19225.825,E2 -19225.825} C_VEL
LIN {X 0,Y 283.992,Z 687.294,A -85,B 0,C 180,E1 -19226.802,E2 -19226.802} C_VEL
LIN {X 0,Y 279.353,Z 699.844,A -85,B 0,C 180,E1 -19228.108,E2 -19228.108} C_VEL
LIN {X 0,Y 274.601,Z 711.241,A -85,B 0,C 180,E1 -19229.637,E2 -19229.637} C_VEL
LIN {X 0,Y 269.229,Z 722.685,A -85,B 0,C 180,E1 -19231.549,E2 -19231.549} C_VEL
LIN {X 0,Y 264.353,Z 732.117,A -85,B 0,C 180,E1 -19233.557,E2 -19233.557} C_VEL
LIN {X 0,Y 259.863,Z 740.098,A -85,B 0,C 180,E1 -19235.642,E2 -19235.642} C_VEL
LIN {X 0,Y 255.254,Z 747.593,A -85,B 0,C 180,E1 -19238.179,E2 -19238.179} C_VEL
LIN {X 0,Y 251.876,Z 752.837,A -85,B 0,C 180,E1 -19240.438,E2 -19240.438} C_VEL
LIN {X 0,Y 247.934,Z 758.225,A -85,B 0,C 180,E1 -19243.533,E2 -19243.533} C_VEL
LIN {X 0,Y 246.243,Z 760.308,A -85,B 0,C 180,E1 -19245.116,E2 -19245.116} C_VEL
LIN {X 0,Y 244.804,Z 761.929,A -85,B 0,C 180,E1 -19246.722,E2 -19246.722} C_VEL
LIN {X 0,Y 242.63,Z 763.995,A -85,B 0,C 180,E1 -19249.991,E2 -19249.991} C_VEL
LIN {X 0,Y 241.015,Z 764.557,A -85,B 0,C 180,E1 -19253.302,E2 -19253.302} C_VEL
LIN {X 0,Y 240.597,Z 764.225,A -85,B 0,C 180,E1 -19254.973,E2 -19254.973} C_VEL
LIN {X 0,Y 240.262,Z 763.483,A -85,B 0,C 180,E1 -19256.646,E2 -19256.646} C_VEL
LIN {X 0,Y 240.055,Z 762.34,A -85,B 0,C 180,E1 -19258.322,E2 -19258.322} C_VEL
LIN {X 0,Y 239.941,Z 760.793,A -85,B 0,C 180,E1 -19260,E2 -19260} C_VEL
LIN {X 0,Y 239.864,Z 757.635,A -85,B 0,C 180,E1 -19262.519,E2 -19262.519} C_VEL
LIN {X 0,Y 239.953,Z 753.054,A -85,B 0,C 180,E1 -19265.23,E2 -19265.23} C_VEL
LIN {X 0,Y 240.271,Z 746.95,A -85,B 0,C 180,E1 -19267.986,E2 -19267.986} C_VEL
LIN {X 0,Y 240.741,Z 739.871,A -85,B 0,C 180,E1 -19270.513,E2 -19270.513} C_VEL
LIN {X 0,Y 241.498,Z 731.163,A -85,B 0,C 180,E1 -19273.034,E2 -19273.034} C_VEL
LIN {X 0,Y 242.352,Z 722.389,A -85,B 0,C 180,E1 -19275.129,E2 -19275.129} C_VEL
LIN {X 0,Y 243.257,Z 712.688,A -85,B 0,C 180,E1 -19277.062,E2 -19277.062} C_VEL
LIN {X 0,Y 244.47,Z 701.656,A -85,B 0,C 180,E1 -19278.87,E2 -19278.87} C_VEL
LIN {X 0,Y 245.716,Z 689.244,A -85,B 0,C 180,E1 -19280.51,E2 -19280.51} C_VEL
LIN {X 0,Y 246.818,Z 675.443,A -85,B 0,C 180,E1 -19281.946,E2 -19281.946} C_VEL
LIN {X 0,Y 247.924,Z 660.51,A -85,B 0,C 180,E1 -19283.106,E2 -19283.106} C_VEL
LIN {X 0,Y 248.981,Z 641.362,A -85,B 0,C 180,E1 -19284.105,E2 -19284.105} C_VEL
LIN {X 0,Y 252.179,Z 580.22,A -85,B 0,C 180,E1 -19286.968,E2 -19286.968} C_VEL
LIN {X 0,Y 249.049,Z 550.663,A -85,B 0,C 180,E1 -19288.601,E2 -19288.601} C_VEL
LIN {X 0,Y 248.201,Z 538.177,A -85,B 0,C 180,E1 -19289.296,E2 -19289.296} C_VEL
LIN {X 0,Y 248.446,Z 535.378,A -85,B 0,C 180,E1 -19290.139,E2 -19290.139} C_VEL
LIN {X 0,Y 245.81,Z 522.501,A -85,B 0,C 180,E1 -19294.367,E2 -19294.367} C_VEL
LIN {X 0,Y 243.031,Z 510.125,A -85,B 0,C 180,E1 -19298.667,E2 -19298.667} C_VEL
LIN {X 0,Y 241.997,Z 505.461,A -85,B 0,C 180,E1 -19300.384,E2 -19300.384} C_VEL
LIN {X 0,Y 241.933,Z 505.473,A -85,B 0,C 180,E1 -19304.202,E2 -19304.202} C_VEL
LIN {X 0,Y 241.939,Z 505.473,A -85,B 0,C 180,E1 -19308.078,E2 -19308.078} C_VEL
LIN {X 0,Y 241.992,Z 505.464,A -85,B 0,C 180,E1 -19312.418,E2 -19312.418} C_VEL
LIN {X 0,Y 241.989,Z 505.463,A -85,B 0,C 180,E1 -19316.508,E2 -19316.508} C_VEL
LIN {X 0,Y 242.038,Z 505.458,A -85,B 0,C 180,E1 -19320.587,E2 -19320.587} C_VEL
LIN {X 0,Y 242.069,Z 505.453,A -85,B 0,C 180,E1 -19324.183,E2 -19324.183} C_VEL
LIN {X 0,Y 242.055,Z 505.457,A -85,B 0,C 180,E1 -19328.297,E2 -19328.297} C_VEL
LIN {X 0,Y 242.165,Z 505.443,A -85,B 0,C 180,E1 -19333.278,E2 -19333.278} C_VEL
LIN {X 0,Y 242.188,Z 505.44,A -85,B 0,C 180,E1 -19338.28,E2 -19338.28} C_VEL
LIN {X 0,Y 242.437,Z 505.41,A -85,B 0,C 180,E1 -19341.666,E2 -19341.666} C_VEL
LIN {X 0,Y 242.264,Z 505.432,A -85,B 0,C 180,E1 -19345.007,E2 -19345.007} C_VEL
LIN {X 0,Y 242.641,Z 505.382,A -85,B 0,C 180,E1 -19348.34,E2 -19348.34} C_VEL
LIN {X 0,Y 242.639,Z 505.386,A -85,B 0,C 180,E1 -19351.66,E2 -19351.66} C_VEL
LIN {X 0,Y 242.435,Z 505.408,A -85,B 0,C 180,E1 -19356.659,E2 -19356.659} C_VEL
LIN {X 0,Y 242.347,Z 505.42,A -85,B 0,C 180,E1 -19360.02,E2 -19360.02} C_VEL
LIN {X 0,Y 242.168,Z 505.444,A -85,B 0,C 180,E1 -19365.141,E2 -19365.141} C_VEL
LIN {X 0,Y 242.075,Z 505.453,A -85,B 0,C 180,E1 -19368.624,E2 -19368.624} C_VEL
LIN {X 0,Y 242.014,Z 505.461,A -85,B 0,C 180,E1 -19372.18,E2 -19372.18} C_VEL
LIN {X 0,Y 242.068,Z 505.454,A -85,B 0,C 180,E1 -19375.838,E2 -19375.838} C_VEL
LIN {X 0,Y 242.008,Z 505.465,A -85,B 0,C 180,E1 -19379.583,E2 -19379.583} C_VEL
LIN {X 0,Y 241.992,Z 505.465,A -85,B 0,C 180,E1 -19383.491,E2 -19383.491} C_VEL
LIN {X 0,Y 242.004,Z 505.465,A -85,B 0,C 180,E1 -19387.579,E2 -19387.579} C_VEL
LIN {X 0,Y 241.945,Z 505.468,A -85,B 0,C 180,E1 -19391.921,E2 -19391.921} C_VEL
LIN {X 0,Y 241.938,Z 505.471,A -85,B 0,C 180,E1 -19396.571,E2 -19396.571} C_VEL
LIN {X 0,Y 241.957,Z 505.469,A -85,B 0,C 180,E1 -19400.281,E2 -19400.281} C_VEL
LIN {X 0,Y 242.082,Z 505.657,A -85,B 0,C 180,E1 -19402.834,E2 -19402.834} C_VEL
LIN {X 0,Y 245.648,Z 521.234,A -85,B 0,C 180,E1 -19406.788,E2 -19406.788} C_VEL
LIN {X 0,Y 248.802,Z 535.821,A -85,B 0,C 180,E1 -19410.375,E2 -19410.375} C_VEL
LIN {X 0,Y 248.633,Z 539.82,A -85,B 0,C 180,E1 -19411.28,E2 -19411.28} C_VEL
LIN {X 0,Y 247.533,Z 550.644,A -85,B 0,C 180,E1 -19413.67,E2 -19413.67} C_VEL
LIN {X 0,Y 249.243,Z 572.209,A -85,B 0,C 180,E1 -19414.782,E2 -19414.782} C_VEL
LIN {X 0,Y 250.41,Z 582.704,A -85,B 0,C 180,E1 -19415.324,E2 -19415.324} C_VEL
LIN {X 0,Y 246.874,Z 662.312,A -85,B 0,C 180,E1 -19418.991,E2 -19418.991} C_VEL
LIN {X 0,Y 246.164,Z 675.235,A -85,B 0,C 180,E1 -19419.856,E2 -19419.856} C_VEL
LIN {X 0,Y 245.153,Z 689.78,A -85,B 0,C 180,E1 -19421.219,E2 -19421.219} C_VEL
LIN {X 0,Y 243.914,Z 702.738,A -85,B 0,C 180,E1 -19422.822,E2 -19422.822} C_VEL
LIN {X 0,Y 243.193,Z 712.255,A -85,B 0,C 180,E1 -19424.281,E2 -19424.281} C_VEL
LIN {X 0,Y 242.249,Z 722.407,A -85,B 0,C 180,E1 -19426.152,E2 -19426.152} C_VEL
LIN {X 0,Y 241.28,Z 733.343,A -85,B 0,C 180,E1 -19428.661,E2 -19428.661} C_VEL
LIN {X 0,Y 240.695,Z 740.801,A -85,B 0,C 180,E1 -19430.759,E2 -19430.759} C_VEL
LIN {X 0,Y 240.265,Z 748.108,A -85,B 0,C 180,E1 -19433.281,E2 -19433.281} C_VEL
LIN {X 0,Y 240.001,Z 753.904,A -85,B 0,C 180,E1 -19435.802,E2 -19435.802} C_VEL
LIN {X 0,Y 239.94,Z 758.427,A -85,B 0,C 180,E1 -19438.322,E2 -19438.322} C_VEL
LIN {X 0,Y 239.916,Z 760.83,A -85,B 0,C 180,E1 -19440,E2 -19440} C_VEL
LIN {X 0,Y 239.973,Z 762.725,A -85,B 0,C 180,E1 -19441.678,E2 -19441.678} C_VEL
LIN {X 0,Y 240.04,Z 764.186,A -85,B 0,C 180,E1 -19443.357,E2 -19443.357} C_VEL
LIN {X 0,Y 240.328,Z 765.338,A -85,B 0,C 180,E1 -19445.302,E2 -19445.302} C_VEL
LIN {X 0,Y 240.023,Z 765.873,A -85,B 0,C 180,E1 -19446.705,E2 -19446.705} C_VEL
LIN {X 0,Y 237.934,Z 766.201,A -85,B 0,C 180,E1 -19449.031,E2 -19449.031} C_VEL
LIN {X 0,Y 236.383,Z 766.073,A -85,B 0,C 180,E1 -19450.916,E2 -19450.916} C_VEL
LIN {X 0,Y 236.188,Z 765.686,A -85,B 0,C 180,E1 -19452.347,E2 -19452.347} C_VEL
LIN {X 0,Y 236.427,Z 765.429,A -85,B 0,C 180,E1 -19452.818,E2 -19452.818} C_VEL
LIN {X 0,Y 238.414,Z 763.749,A -85,B 0,C 180,E1 -19455.385,E2 -19455.385} C_VEL
LIN {X 0,Y 240.767,Z 761.134,A -85,B 0,C 180,E1 -19457.848,E2 -19457.848} C_VEL
LIN {X 0,Y 243.739,Z 757.522,A -85,B 0,C 180,E1 -19460.244,E2 -19460.244} C_VEL
LIN {X 0,Y 247.17,Z 752.849,A -85,B 0,C 180,E1 -19462.573,E2 -19462.573} C_VEL
LIN {X 0,Y 251.75,Z 745.951,A -85,B 0,C 180,E1 -19465.197,E2 -19465.197} C_VEL
LIN {X 0,Y 256.939,Z 737.266,A -85,B 0,C 180,E1 -19467.71,E2 -19467.71} C_VEL
LIN {X 0,Y 261.831,Z 727.988,A -85,B 0,C 180,E1 -19469.774,E2 -19469.774} C_VEL
LIN {X 0,Y 266.646,Z 717.848,A -85,B 0,C 180,E1 -19471.591,E2 -19471.591} C_VEL
LIN {X 0,Y 271.921,Z 705.197,A -85,B 0,C 180,E1 -19473.314,E2 -19473.314} C_VEL
LIN {X 0,Y 276.001,Z 693.873,A -85,B 0,C 180,E1 -19474.511,E2 -19474.511} C_VEL
LIN {X 0,Y 279.712,Z 681.628,A -85,B 0,C 180,E1 -19475.523,E2 -19475.523} C_VEL
LIN {X 0,Y 283.045,Z 668.235,A -85,B 0,C 180,E1 -19476.357,E2 -19476.357} C_VEL
LIN {X 0,Y 295.786,Z 605.538,A -85,B 0,C 180,E1 -19479.225,E2 -19479.225} C_VEL
LIN {X 0,Y 296.209,Z 601.114,A -85,B 0,C 180,E1 -19479.882,E2 -19479.882} C_VEL
LIN {X 0,Y 295.719,Z 597.937,A -85,B 0,C 180,E1 -19481.278,E2 -19481.278} C_VEL
LIN {X 0,Y 295.436,Z 595.277,A -85,B 0,C 180,E1 -19482.896,E2 -19482.896} C_VEL
LIN {X 0,Y 295.424,Z 593.718,A -85,B 0,C 180,E1 -19484.978,E2 -19484.978} C_VEL
LIN {X 0,Y 295.779,Z 593.458,A -85,B 0,C 180,E1 -19486.443,E2 -19486.443} C_VEL
LIN {X 0,Y 296.834,Z 594.253,A -85,B 0,C 180,E1 -19488.59,E2 -19488.59} C_VEL
LIN {X 0,Y 297.048,Z 594.465,A -85,B 0,C 180,E1 -19488.88,E2 -19488.88} C_VEL
LIN {X 0,Y 281.339,Z 668.889,A -85,B 0,C 180,E1 -19492.433,E2 -19492.433} C_VEL
LIN {X 0,Y 277.788,Z 683.843,A -85,B 0,C 180,E1 -19493.294,E2 -19493.294} C_VEL
LIN {X 0,Y 273.867,Z 696.835,A -85,B 0,C 180,E1 -19494.281,E2 -19494.281} C_VEL
LIN {X 0,Y 269.7,Z 708.756,A -85,B 0,C 180,E1 -19495.474,E2 -19495.474} C_VEL
LIN {X 0,Y 264.361,Z 722.008,A -85,B 0,C 180,E1 -19497.203,E2 -19497.203} C_VEL
LIN {X 0,Y 259.461,Z 732.806,A -85,B 0,C 180,E1 -19499.026,E2 -19499.026} C_VEL
LIN {X 0,Y 254.481,Z 742.711,A -85,B 0,C 180,E1 -19501.099,E2 -19501.099} C_VEL
LIN {X 0,Y 249.353,Z 752.114,A -85,B 0,C 180,E1 -19503.646,E2 -19503.646} C_VEL
LIN {X 0,Y 244.98,Z 759.681,A -85,B 0,C 180,E1 -19506.32,E2 -19506.32} C_VEL
LIN {X 0,Y 241.472,Z 765.36,A -85,B 0,C 180,E1 -19508.884,E2 -19508.884} C_VEL
LIN {X 0,Y 238.267,Z 770.356,A -85,B 0,C 180,E1 -19511.958,E2 -19511.958} C_VEL
LIN {X 0,Y 236.171,Z 773.323,A -85,B 0,C 180,E1 -19514.465,E2 -19514.465} C_VEL
LIN {X 0,Y 234.279,Z 775.871,A -85,B 0,C 180,E1 -19517.878,E2 -19517.878} C_VEL
LIN {X 0,Y 233.616,Z 776.577,A -85,B 0,C 180,E1 -19519.601,E2 -19519.601} C_VEL
LIN {X 0,Y 233.188,Z 776.876,A -85,B 0,C 180,E1 -19521.333,E2 -19521.333} C_VEL
LIN {X 0,Y 232.818,Z 776.246,A -85,B 0,C 180,E1 -19524.804,E2 -19524.804} C_VEL
LIN {X 0,Y 232.903,Z 775.348,A -85,B 0,C 180,E1 -19526.54,E2 -19526.54} C_VEL
LIN {X 0,Y 232.967,Z 773.117,A -85,B 0,C 180,E1 -19529.352,E2 -19529.352} C_VEL
LIN {X 0,Y 232.861,Z 775.225,A -85,B 0,C 180,E1 -19531.73,E2 -19531.73} C_VEL
LIN {X 0,Y 232.873,Z 776.311,A -85,B 0,C 180,E1 -19533.461,E2 -19533.461} C_VEL
LIN {X 0,Y 232.877,Z 777.369,A -85,B 0,C 180,E1 -19536.934,E2 -19536.934} C_VEL
LIN {X 0,Y 233.513,Z 777.043,A -85,B 0,C 180,E1 -19540.404,E2 -19540.404} C_VEL
LIN {X 0,Y 234.867,Z 775.38,A -85,B 0,C 180,E1 -19543.851,E2 -19543.851} C_VEL
LIN {X 0,Y 237.241,Z 772.377,A -85,B 0,C 180,E1 -19547.232,E2 -19547.232} C_VEL
LIN {X 0,Y 240.446,Z 767.76,A -85,B 0,C 180,E1 -19550.719,E2 -19550.719} C_VEL
LIN {X 0,Y 244.195,Z 762.199,A -85,B 0,C 180,E1 -19553.761,E2 -19553.761} C_VEL
LIN {X 0,Y 249.117,Z 754.778,A -85,B 0,C 180,E1 -19556.833,E2 -19556.833} C_VEL
LIN {X 0,Y 254.126,Z 746.691,A -85,B 0,C 180,E1 -19559.399,E2 -19559.399} C_VEL
LIN {X 0,Y 259.806,Z 736.995,A -85,B 0,C 180,E1 -19561.837,E2 -19561.837} C_VEL
LIN {X 0,Y 265.205,Z 726.971,A -85,B 0,C 180,E1 -19563.815,E2 -19563.815} C_VEL
LIN {X 0,Y 271.075,Z 715.185,A -85,B 0,C 180,E1 -19565.686,E2 -19565.686} C_VEL
LIN {X 0,Y 276.792,Z 702.002,A -85,B 0,C 180,E1 -19567.316,E2 -19567.316} C_VEL
LIN {X 0,Y 281.356,Z 690.451,A -85,B 0,C 180,E1 -19568.415,E2 -19568.415} C_VEL
LIN {X 0,Y 286.036,Z 676.351,A -85,B 0,C 180,E1 -19569.477,E2 -19569.477} C_VEL
LIN {X 0,Y 290.649,Z 659.252,A -85,B 0,C 180,E1 -19570.417,E2 -19570.417} C_VEL
LIN {X 0,Y 302.211,Z 605.113,A -85,B 0,C 180,E1 -19572.699,E2 -19572.699} C_VEL
LIN {X 0,Y 302.309,Z 604.402,A -85,B 0,C 180,E1 -19572.785,E2 -19572.785} C_VEL
LIN {X 0,Y 301.433,Z 602.165,A -85,B 0,C 180,E1 -19574.752,E2 -19574.752} C_VEL
LIN {X 0,Y 300.908,Z 602.163,A -85,B 0,C 180,E1 -19577.365,E2 -19577.365} C_VEL
LIN {X 0,Y 300.975,Z 603.034,A -85,B 0,C 180,E1 -19578.628,E2 -19578.628} C_VEL
LIN {X 0,Y 301.49,Z 606.536,A -85,B 0,C 180,E1 -19580.823,E2 -19580.823} C_VEL
LIN {X 0,Y 301.545,Z 607.429,A -85,B 0,C 180,E1 -19581.114,E2 -19581.114} C_VEL
LIN {X 0,Y 289.322,Z 661.803,A -85,B 0,C 180,E1 -19583.602,E2 -19583.602} C_VEL
LIN {X 0,Y 285.444,Z 675.246,A -85,B 0,C 180,E1 -19584.432,E2 -19584.432} C_VEL
LIN {X 0,Y 281.443,Z 686.932,A -85,B 0,C 180,E1 -19585.382,E2 -19585.382} C_VEL
LIN {X 0,Y 276.526,Z 699.417,A -85,B 0,C 180,E1 -19586.66,E2 -19586.66} C_VEL
LIN {X 0,Y 270.952,Z 711.863,A -85,B 0,C 180,E1 -19588.315,E2 -19588.315} C_VEL
LIN {X 0,Y 265.264,Z 723.104,A -85,B 0,C 180,E1 -19590.213,E2 -19590.213} C_VEL
LIN {X 0,Y 259.23,Z 733.873,A -85,B 0,C 180,E1 -19592.555,E2 -19592.555} C_VEL
LIN {X 0,Y 253.703,Z 742.612,A -85,B 0,C 180,E1 -19595.011,E2 -19595.011} C_VEL
LIN {X 0,Y 248.928,Z 749.712,A -85,B 0,C 180,E1 -19597.595,E2 -19597.595} C_VEL
LIN {X 0,Y 244.262,Z 755.92,A -85,B 0,C 180,E1 -19600.678,E2 -19600.678} C_VEL
LIN {X 0,Y 241.249,Z 759.491,A -85,B 0,C 180,E1 -19603.063,E2 -19603.063} C_VEL
LIN {X 0,Y 237.972,Z 762.807,A -85,B 0,C 180,E1 -19606.334,E2 -19606.334} C_VEL
LIN {X 0,Y 236.799,Z 763.88,A -85,B 0,C 180,E1 -19608.009,E2 -19608.009} C_VEL
LIN {X 0,Y 235.45,Z 764.653,A -85,B 0,C 180,E1 -19610.074,E2 -19610.074} C_VEL
LIN {X 0,Y 233.974,Z 764.765,A -85,B 0,C 180,E1 -19613.099,E2 -19613.099} C_VEL
LIN {X 0,Y 233.186,Z 763.41,A -85,B 0,C 180,E1 -19616.544,E2 -19616.544} C_VEL
LIN {X 0,Y 232.968,Z 762.152,A -85,B 0,C 180,E1 -19618.271,E2 -19618.271} C_VEL
LIN {X 0,Y 232.834,Z 759.424,A -85,B 0,C 180,E1 -19620.865,E2 -19620.865} C_VEL
LIN {X 0,Y 232.799,Z 755.673,A -85,B 0,C 180,E1 -19623.461,E2 -19623.461} C_VEL
LIN {X 0,Y 232.97,Z 750.809,A -85,B 0,C 180,E1 -19626.061,E2 -19626.061} C_VEL
LIN {X 0,Y 233.299,Z 744.688,A -85,B 0,C 180,E1 -19628.663,E2 -19628.663} C_VEL
LIN {X 0,Y 233.85,Z 737.069,A -85,B 0,C 180,E1 -19631.265,E2 -19631.265} C_VEL
LIN {X 0,Y 234.75,Z 727.636,A -85,B 0,C 180,E1 -19633.857,E2 -19633.857} C_VEL
LIN {X 0,Y 235.572,Z 718.07,A -85,B 0,C 180,E1 -19636.019,E2 -19636.019} C_VEL
LIN {X 0,Y 236.896,Z 706.379,A -85,B 0,C 180,E1 -19638.179,E2 -19638.179} C_VEL
LIN {X 0,Y 238.185,Z 693.743,A -85,B 0,C 180,E1 -19640.06,E2 -19640.06} C_VEL
LIN {X 0,Y 239.403,Z 680.267,A -85,B 0,C 180,E1 -19641.641,E2 -19641.641} C_VEL
LIN {X 0,Y 240.452,Z 666.399,A -85,B 0,C 180,E1 -19642.899,E2 -19642.899} C_VEL
LIN {X 0,Y 241.474,Z 651.254,A -85,B 0,C 180,E1 -19643.875,E2 -19643.875} C_VEL
LIN {X 0,Y 245.242,Z 580.887,A -85,B 0,C 180,E1 -19647.292,E2 -19647.292} C_VEL
LIN {X 0,Y 242.155,Z 550.762,A -85,B 0,C 180,E1 -19649.015,E2 -19649.015} C_VEL
LIN {X 0,Y 241.345,Z 538.126,A -85,B 0,C 180,E1 -19649.733,E2 -19649.733} C_VEL
LIN {X 0,Y 241.226,Z 535.222,A -85,B 0,C 180,E1 -19650.654,E2 -19650.654} C_VEL
LIN {X 0,Y 238.689,Z 523.116,A -85,B 0,C 180,E1 -19654.752,E2 -19654.752} C_VEL
LIN {X 0,Y 236.238,Z 512.126,A -85,B 0,C 180,E1 -19658.663,E2 -19658.663} C_VEL
LIN {X 0,Y 234.925,Z 506.342,A -85,B 0,C 180,E1 -19660.875,E2 -19660.875} C_VEL
LIN {X 0,Y 234.897,Z 506.35,A -85,B 0,C 180,E1 -19664.104,E2 -19664.104} C_VEL
LIN {X 0,Y 234.885,Z 506.351,A -85,B 0,C 180,E1 -19668.832,E2 -19668.832} C_VEL
LIN {X 0,Y 234.919,Z 506.347,A -85,B 0,C 180,E1 -19671.079,E2 -19671.079} C_VEL
LIN {X 0,Y 234.943,Z 506.343,A -85,B 0,C 180,E1 -19675.364,E2 -19675.364} C_VEL
LIN {X 0,Y 234.933,Z 506.347,A -85,B 0,C 180,E1 -19679.432,E2 -19679.432} C_VEL
LIN {X 0,Y 234.996,Z 506.335,A -85,B 0,C 180,E1 -19683.793,E2 -19683.793} C_VEL
LIN {X 0,Y 235.013,Z 506.335,A -85,B 0,C 180,E1 -19688.97,E2 -19688.97} C_VEL
LIN {X 0,Y 235.098,Z 506.321,A -85,B 0,C 180,E1 -19693.059,E2 -19693.059} C_VEL
LIN {X 0,Y 235.148,Z 506.318,A -85,B 0,C 180,E1 -19697.924,E2 -19697.924} C_VEL
LIN {X 0,Y 235.392,Z 506.287,A -85,B 0,C 180,E1 -19701.414,E2 -19701.414} C_VEL
LIN {X 0,Y 235.408,Z 506.285,A -85,B 0,C 180,E1 -19703.141,E2 -19703.141} C_VEL
LIN {X 0,Y 235.6,Z 506.259,A -85,B 0,C 180,E1 -19708.29,E2 -19708.29} C_VEL
LIN {X 0,Y 235.598,Z 506.263,A -85,B 0,C 180,E1 -19711.709,E2 -19711.709} C_VEL
LIN {X 0,Y 235.407,Z 506.284,A -85,B 0,C 180,E1 -19716.858,E2 -19716.858} C_VEL
LIN {X 0,Y 235.255,Z 506.303,A -85,B 0,C 180,E1 -19720.326,E2 -19720.326} C_VEL
LIN {X 0,Y 235.115,Z 506.321,A -85,B 0,C 180,E1 -19725.606,E2 -19725.606} C_VEL
LIN {X 0,Y 235.01,Z 506.336,A -85,B 0,C 180,E1 -19729.205,E2 -19729.205} C_VEL
LIN {X 0,Y 234.962,Z 506.341,A -85,B 0,C 180,E1 -19732.883,E2 -19732.883} C_VEL
LIN {X 0,Y 234.969,Z 506.338,A -85,B 0,C 180,E1 -19736.657,E2 -19736.657} C_VEL
LIN {X 0,Y 234.924,Z 506.345,A -85,B 0,C 180,E1 -19740.569,E2 -19740.569} C_VEL
LIN {X 0,Y 234.961,Z 506.338,A -85,B 0,C 180,E1 -19744.633,E2 -19744.633} C_VEL
LIN {X 0,Y 234.943,Z 506.344,A -85,B 0,C 180,E1 -19748.944,E2 -19748.944} C_VEL
LIN {X 0,Y 234.891,Z 506.351,A -85,B 0,C 180,E1 -19753.485,E2 -19753.485} C_VEL
LIN {X 0,Y 234.891,Z 506.349,A -85,B 0,C 180,E1 -19756.515,E2 -19756.515} C_VEL
LIN {X 0,Y 234.92,Z 506.349,A -85,B 0,C 180,E1 -19761.079,E2 -19761.079} C_VEL
LIN {X 0,Y 234.991,Z 506.453,A -85,B 0,C 180,E1 -19762.413,E2 -19762.413} C_VEL
LIN {X 0,Y 238.475,Z 521.665,A -85,B 0,C 180,E1 -19766.36,E2 -19766.36} C_VEL
LIN {X 0,Y 241.796,Z 536.777,A -85,B 0,C 180,E1 -19770.149,E2 -19770.149} C_VEL
LIN {X 0,Y 241.749,Z 539.796,A -85,B 0,C 180,E1 -19770.847,E2 -19770.847} C_VEL
LIN {X 0,Y 240.566,Z 550.953,A -85,B 0,C 180,E1 -19773.339,E2 -19773.339} C_VEL
LIN {X 0,Y 242.365,Z 573.645,A -85,B 0,C 180,E1 -19774.537,E2 -19774.537} C_VEL
LIN {X 0,Y 243.379,Z 583.519,A -85,B 0,C 180,E1 -19775.06,E2 -19775.06} C_VEL
LIN {X 0,Y 239.863,Z 661.068,A -85,B 0,C 180,E1 -19778.797,E2 -19778.797} C_VEL
LIN {X 0,Y 239.072,Z 675.392,A -85,B 0,C 180,E1 -19779.776,E2 -19779.776} C_VEL
LIN {X 0,Y 238.121,Z 688.788,A -85,B 0,C 180,E1 -19781.055,E2 -19781.055} C_VEL
LIN {X 0,Y 237.031,Z 700.806,A -85,B 0,C 180,E1 -19782.53,E2 -19782.53} C_VEL
LIN {X 0,Y 236.122,Z 711.892,A -85,B 0,C 180,E1 -19784.241,E2 -19784.241} C_VEL
LIN {X 0,Y 235.161,Z 722.137,A -85,B 0,C 180,E1 -19786.167,E2 -19786.167} C_VEL
LIN {X 0,Y 234.329,Z 731.523,A -85,B 0,C 180,E1 -19788.32,E2 -19788.32} C_VEL
LIN {X 0,Y 233.612,Z 740.65,A -85,B 0,C 180,E1 -19790.913,E2 -19790.913} C_VEL
LIN {X 0,Y 233.178,Z 748.103,A -85,B 0,C 180,E1 -19793.554,E2 -19793.554} C_VEL
LIN {X 0,Y 232.949,Z 754.707,A -85,B 0,C 180,E1 -19796.541,E2 -19796.541} C_VEL
LIN {X 0,Y 232.836,Z 759.105,A -85,B 0,C 180,E1 -19799.135,E2 -19799.135} C_VEL
LIN {X 0,Y 232.907,Z 762.375,A -85,B 0,C 180,E1 -19801.729,E2 -19801.729} C_VEL
LIN {X 0,Y 232.969,Z 763.984,A -85,B 0,C 180,E1 -19803.459,E2 -19803.459} C_VEL
LIN {X 0,Y 233.69,Z 765.926,A -85,B 0,C 180,E1 -19806.909,E2 -19806.909} C_VEL
LIN {X 0,Y 234.263,Z 766.31,A -85,B 0,C 180,E1 -19808.627,E2 -19808.627} C_VEL
LIN {X 0,Y 234.954,Z 766.272,A -85,B 0,C 180,E1 -19810.339,E2 -19810.339} C_VEL
LIN {X 0,Y 236.427,Z 765.429,A -85,B 0,C 180,E1 -19812.818,E2 -19812.818} C_VEL
LIN {X 0,Y 236.427,Z 765.037,A -85,B 0,C 180,E1 -19813.781,E2 -19813.781} C_VEL
LIN {X 0,Y 233.251,Z 763.605,A -85,B 0,C 180,E1 -19816.97,E2 -19816.97} C_VEL
LIN {X 0,Y 233.564,Z 762.745,A -85,B 0,C 180,E1 -19817.918,E2 -19817.918} C_VEL
LIN {X 0,Y 237.236,Z 758.988,A -85,B 0,C 180,E1 -19820.824,E2 -19820.824} C_VEL
LIN {X 0,Y 240.845,Z 754.687,A -85,B 0,C 180,E1 -19823.2,E2 -19823.2} C_VEL
LIN {X 0,Y 246.376,Z 747.234,A -85,B 0,C 180,E1 -19826.241,E2 -19826.241} C_VEL
LIN {X 0,Y 251.865,Z 738.805,A -85,B 0,C 180,E1 -19828.773,E2 -19828.773} C_VEL
LIN {X 0,Y 257.039,Z 730,A -85,B 0,C 180,E1 -19830.842,E2 -19830.842} C_VEL
LIN {X 0,Y 262.571,Z 719.248,A -85,B 0,C 180,E1 -19832.821,E2 -19832.821} C_VEL
LIN {X 0,Y 267.624,Z 708.207,A -85,B 0,C 180,E1 -19834.375,E2 -19834.375} C_VEL
LIN {X 0,Y 272.429,Z 696.161,A -85,B 0,C 180,E1 -19835.709,E2 -19835.709} C_VEL
LIN {X 0,Y 276.871,Z 682.653,A -85,B 0,C 180,E1 -19836.848,E2 -19836.848} C_VEL
LIN {X 0,Y 280.511,Z 669.077,A -85,B 0,C 180,E1 -19837.697,E2 -19837.697} C_VEL
LIN {X 0,Y 293.722,Z 608.101,A -85,B 0,C 180,E1 -19840.474,E2 -19840.474} C_VEL
LIN {X 0,Y 293.877,Z 606.527,A -85,B 0,C 180,E1 -19840.744,E2 -19840.744} C_VEL
LIN {X 0,Y 293.669,Z 603.988,A -85,B 0,C 180,E1 -19841.9,E2 -19841.9} C_VEL
LIN {X 0,Y 293.532,Z 601.644,A -85,B 0,C 180,E1 -19843.501,E2 -19843.501} C_VEL
LIN {X 0,Y 293.621,Z 600.582,A -85,B 0,C 180,E1 -19845.052,E2 -19845.052} C_VEL
LIN {X 0,Y 294.16,Z 600.424,A -85,B 0,C 180,E1 -19847.007,E2 -19847.007} C_VEL
LIN {X 0,Y 294.571,Z 600.645,A -85,B 0,C 180,E1 -19847.787,E2 -19847.787} C_VEL
LIN {X 0,Y 277.493,Z 676.296,A -85,B 0,C 180,E1 -19851.415,E2 -19851.415} C_VEL
LIN {X 0,Y 273.302,Z 690.665,A -85,B 0,C 180,E1 -19852.357,E2 -19852.357} C_VEL
LIN {X 0,Y 268.713,Z 703.649,A -85,B 0,C 180,E1 -19853.486,E2 -19853.486} C_VEL
LIN {X 0,Y 263.395,Z 716.533,A -85,B 0,C 180,E1 -19854.993,E2 -19854.993} C_VEL
LIN {X 0,Y 258.43,Z 727.203,A -85,B 0,C 180,E1 -19856.585,E2 -19856.585} C_VEL
LIN {X 0,Y 252.9,Z 737.856,A -85,B 0,C 180,E1 -19858.597,E2 -19858.597} C_VEL
LIN {X 0,Y 247.843,Z 746.728,A -85,B 0,C 180,E1 -19860.715,E2 -19860.715} C_VEL
LIN {X 0,Y 243.243,Z 754.15,A -85,B 0,C 180,E1 -19862.931,E2 -19862.931} C_VEL
LIN {X 0,Y 238.643,Z 761.19,A -85,B 0,C 180,E1 -19865.651,E2 -19865.651} C_VEL
LIN {X 0,Y 235.06,Z 766.25,A -85,B 0,C 180,E1 -19868.172,E2 -19868.172} C_VEL
LIN {X 0,Y 231.575,Z 771.065,A -85,B 0,C 180,E1 -19871.418,E2 -19871.418} C_VEL
LIN {X 0,Y 229.345,Z 773.727,A -85,B 0,C 180,E1 -19873.991,E2 -19873.991} C_VEL
LIN {X 0,Y 228.192,Z 775.036,A -85,B 0,C 180,E1 -19875.736,E2 -19875.736} C_VEL
LIN {X 0,Y 226.613,Z 776.448,A -85,B 0,C 180,E1 -19879.276,E2 -19879.276} C_VEL
LIN {X 0,Y 225.855,Z 776.346,A -85,B 0,C 180,E1 -19882.85,E2 -19882.85} C_VEL
LIN {X 0,Y 225.742,Z 775.487,A -85,B 0,C 180,E1 -19885.04,E2 -19885.04} C_VEL
LIN {X 0,Y 225.839,Z 774.629,A -85,B 0,C 180,E1 -19886.432,E2 -19886.432} C_VEL
LIN {X 0,Y 225.931,Z 772.133,A -85,B 0,C 180,E1 -19889.276,E2 -19889.276} C_VEL
LIN {X 0,Y 225.806,Z 774.444,A -85,B 0,C 180,E1 -19891.784,E2 -19891.784} C_VEL
LIN {X 0,Y 225.732,Z 776.298,A -85,B 0,C 180,E1 -19894.932,E2 -19894.932} C_VEL
LIN {X 0,Y 225.806,Z 776.931,A -85,B 0,C 180,E1 -19897.152,E2 -19897.152} C_VEL
LIN {X 0,Y 226.515,Z 776.872,A -85,B 0,C 180,E1 -19900.729,E2 -19900.729} C_VEL
LIN {X 0,Y 227.954,Z 775.493,A -85,B 0,C 180,E1 -19904.279,E2 -19904.279} C_VEL
LIN {X 0,Y 230.476,Z 772.808,A -85,B 0,C 180,E1 -19907.754,E2 -19907.754} C_VEL
LIN {X 0,Y 233.751,Z 768.68,A -85,B 0,C 180,E1 -19911.243,E2 -19911.243} C_VEL
LIN {X 0,Y 237.804,Z 763.343,A -85,B 0,C 180,E1 -19914.441,E2 -19914.441} C_VEL
LIN {X 0,Y 242.957,Z 756.3,A -85,B 0,C 180,E1 -19917.57,E2 -19917.57} C_VEL
LIN {X 0,Y 249.013,Z 747.565,A -85,B 0,C 180,E1 -19920.532,E2 -19920.532} C_VEL
LIN {X 0,Y 254.998,Z 738.145,A -85,B 0,C 180,E1 -19922.979,E2 -19922.979} C_VEL
LIN {X 0,Y 260.683,Z 728.574,A -85,B 0,C 180,E1 -19924.953,E2 -19924.953} C_VEL
LIN {X 0,Y 267.334,Z 716.152,A -85,B 0,C 180,E1 -19926.968,E2 -19926.968} C_VEL
LIN {X 0,Y 273.345,Z 703.482,A -85,B 0,C 180,E1 -19928.572,E2 -19928.572} C_VEL
LIN {X 0,Y 278.71,Z 690.747,A -85,B 0,C 180,E1 -19929.782,E2 -19929.782} C_VEL
LIN {X 0,Y 283.608,Z 677.155,A -85,B 0,C 180,E1 -19930.813,E2 -19930.813} C_VEL
LIN {X 0,Y 288.253,Z 661.038,A -85,B 0,C 180,E1 -19931.694,E2 -19931.694} C_VEL
LIN {X 0,Y 299.892,Z 610.144,A -85,B 0,C 180,E1 -19933.84,E2 -19933.84} C_VEL
LIN {X 0,Y 299.63,Z 609.092,A -85,B 0,C 180,E1 -19934.722,E2 -19934.722} C_VEL
LIN {X 0,Y 299.099,Z 609.051,A -85,B 0,C 180,E1 -19937.462,E2 -19937.462} C_VEL
LIN {X 0,Y 299.111,Z 609.879,A -85,B 0,C 180,E1 -19938.471,E2 -19938.471} C_VEL
LIN {X 0,Y 299.283,Z 612.254,A -85,B 0,C 180,E1 -19939.975,E2 -19939.975} C_VEL
LIN {X 0,Y 287.524,Z 661.772,A -85,B 0,C 180,E1 -19942.222,E2 -19942.222} C_VEL
LIN {X 0,Y 284.069,Z 673.121,A -85,B 0,C 180,E1 -19942.883,E2 -19942.883} C_VEL
LIN {X 0,Y 279.688,Z 685.595,A -85,B 0,C 180,E1 -19943.819,E2 -19943.819} C_VEL
LIN {X 0,Y 273.854,Z 699.537,A -85,B 0,C 180,E1 -19945.225,E2 -19945.225} C_VEL
LIN {X 0,Y 268.077,Z 711.733,A -85,B 0,C 180,E1 -19946.82,E2 -19946.82} C_VEL
LIN {X 0,Y 261.526,Z 723.714,A -85,B 0,C 180,E1 -19948.848,E2 -19948.848} C_VEL
LIN {X 0,Y 255.969,Z 732.984,A -85,B 0,C 180,E1 -19950.833,E2 -19950.833} C_VEL
LIN {X 0,Y 250.008,Z 741.859,A -85,B 0,C 180,E1 -19953.27,E2 -19953.27} C_VEL
LIN {X 0,Y 245.391,Z 748.14,A -85,B 0,C 180,E1 -19955.463,E2 -19955.463} C_VEL
LIN {X 0,Y 240.09,Z 754.822,A -85,B 0,C 180,E1 -19958.537,E2 -19958.537} C_VEL
LIN {X 0,Y 236.662,Z 758.636,A -85,B 0,C 180,E1 -19960.934,E2 -19960.934} C_VEL
LIN {X 0,Y 232.717,Z 762.405,A -85,B 0,C 180,E1 -19964.229,E2 -19964.229} C_VEL
LIN {X 0,Y 229.882,Z 764.521,A -85,B 0,C 180,E1 -19967.643,E2 -19967.643} C_VEL
LIN {X 0,Y 227.734,Z 765.182,A -85,B 0,C 180,E1 -19971.124,E2 -19971.124} C_VEL
LIN {X 0,Y 226.449,Z 764.32,A -85,B 0,C 180,E1 -19974.658,E2 -19974.658} C_VEL
LIN {X 0,Y 226.113,Z 763.275,A -85,B 0,C 180,E1 -19976.436,E2 -19976.436} C_VEL
LIN {X 0,Y 225.905,Z 761.831,A -85,B 0,C 180,E1 -19978.217,E2 -19978.217} C_VEL
LIN {X 0,Y 225.77,Z 758.905,A -85,B 0,C 180,E1 -19980.892,E2 -19980.892} C_VEL
LIN {X 0,Y 225.723,Z 754.089,A -85,B 0,C 180,E1 -19984.047,E2 -19984.047} C_VEL
LIN {X 0,Y 226.04,Z 747.796,A -85,B 0,C 180,E1 -19987.144,E2 -19987.144} C_VEL
LIN {X 0,Y 226.474,Z 740.885,A -85,B 0,C 180,E1 -19989.827,E2 -19989.827} C_VEL
LIN {X 0,Y 227.144,Z 732.335,A -85,B 0,C 180,E1 -19992.509,E2 -19992.509} C_VEL
LIN {X 0,Y 228.013,Z 723.772,A -85,B 0,C 180,E1 -19994.731,E2 -19994.731} C_VEL
LIN {X 0,Y 228.946,Z 713.375,A -85,B 0,C 180,E1 -19996.955,E2 -19996.955} C_VEL
LIN {X 0,Y 230.226,Z 702.097,A -85,B 0,C 180,E1 -19998.926,E2 -19998.926} C_VEL
LIN {X 0,Y 231.643,Z 688.121,A -85,B 0,C 180,E1 -20000.885,E2 -20000.885} C_VEL
LIN {X 0,Y 232.836,Z 674.061,A -85,B 0,C 180,E1 -20002.4,E2 -20002.4} C_VEL
LIN {X 0,Y 233.876,Z 660.348,A -85,B 0,C 180,E1 -20003.522,E2 -20003.522} C_VEL
LIN {X 0,Y 235.048,Z 639.623,A -85,B 0,C 180,E1 -20004.687,E2 -20004.687} C_VEL
LIN {X 0,Y 238.352,Z 581.734,A -85,B 0,C 180,E1 -20007.63,E2 -20007.63} C_VEL
LIN {X 0,Y 235.346,Z 552.091,A -85,B 0,C 180,E1 -20009.371,E2 -20009.371} C_VEL
LIN {X 0,Y 234.422,Z 538.069,A -85,B 0,C 180,E1 -20010.176,E2 -20010.176} C_VEL
LIN {X 0,Y 232.569,Z 528.442,A -85,B 0,C 180,E1 -20013.47,E2 -20013.47} C_VEL
LIN {X 0,Y 229.87,Z 516.006,A -85,B 0,C 180,E1 -20017.949,E2 -20017.949} C_VEL
LIN {X 0,Y 227.865,Z 507.224,A -85,B 0,C 180,E1 -20021.338,E2 -20021.338} C_VEL
LIN {X 0,Y 227.835,Z 507.23,A -85,B 0,C 180,E1 -20025.192,E2 -20025.192} C_VEL
LIN {X 0,Y 227.827,Z 507.233,A -85,B 0,C 180,E1 -20029.623,E2 -20029.623} C_VEL
LIN {X 0,Y 227.884,Z 507.221,A -85,B 0,C 180,E1 -20034.129,E2 -20034.129} C_VEL
LIN {X 0,Y 227.873,Z 507.223,A -85,B 0,C 180,E1 -20038.378,E2 -20038.378} C_VEL
LIN {X 0,Y 227.888,Z 507.22,A -85,B 0,C 180,E1 -20042.445,E2 -20042.445} C_VEL
LIN {X 0,Y 227.916,Z 507.217,A -85,B 0,C 180,E1 -20046.367,E2 -20046.367} C_VEL
LIN {X 0,Y 227.944,Z 507.214,A -85,B 0,C 180,E1 -20050.175,E2 -20050.175} C_VEL
LIN {X 0,Y 228.059,Z 507.2,A -85,B 0,C 180,E1 -20053.898,E2 -20053.898} C_VEL
LIN {X 0,Y 228.173,Z 507.189,A -85,B 0,C 180,E1 -20059.35,E2 -20059.35} C_VEL
LIN {X 0,Y 228.36,Z 507.162,A -85,B 0,C 180,E1 -20062.929,E2 -20062.929} C_VEL
LIN {X 0,Y 228.559,Z 507.136,A -85,B 0,C 180,E1 -20068.238,E2 -20068.238} C_VEL
LIN {X 0,Y 228.557,Z 507.139,A -85,B 0,C 180,E1 -20071.762,E2 -20071.762} C_VEL
LIN {X 0,Y 228.36,Z 507.163,A -85,B 0,C 180,E1 -20077.071,E2 -20077.071} C_VEL
LIN {X 0,Y 228.173,Z 507.185,A -85,B 0,C 180,E1 -20080.65,E2 -20080.65} C_VEL
LIN {X 0,Y 228.059,Z 507.197,A -85,B 0,C 180,E1 -20086.102,E2 -20086.102} C_VEL
LIN {X 0,Y 227.944,Z 507.216,A -85,B 0,C 180,E1 -20089.825,E2 -20089.825} C_VEL
LIN {X 0,Y 227.915,Z 507.218,A -85,B 0,C 180,E1 -20093.632,E2 -20093.632} C_VEL
LIN {X 0,Y 227.88,Z 507.225,A -85,B 0,C 180,E1 -20097.556,E2 -20097.556} C_VEL
LIN {X 0,Y 227.87,Z 507.224,A -85,B 0,C 180,E1 -20101.622,E2 -20101.622} C_VEL
LIN {X 0,Y 227.901,Z 507.22,A -85,B 0,C 180,E1 -20105.868,E2 -20105.868} C_VEL
LIN {X 0,Y 227.835,Z 507.227,A -85,B 0,C 180,E1 -20110.375,E2 -20110.375} C_VEL
LIN {X 0,Y 227.837,Z 507.23,A -85,B 0,C 180,E1 -20115.192,E2 -20115.192} C_VEL
LIN {X 0,Y 227.827,Z 507.232,A -85,B 0,C 180,E1 -20119.624,E2 -20119.624} C_VEL
LIN {X 0,Y 227.935,Z 507.316,A -85,B 0,C 180,E1 -20121.998,E2 -20121.998} C_VEL
LIN {X 0,Y 231.512,Z 522.971,A -85,B 0,C 180,E1 -20126.151,E2 -20126.151} C_VEL
LIN {X 0,Y 234.791,Z 537.837,A -85,B 0,C 180,E1 -20129.956,E2 -20129.956} C_VEL
LIN {X 0,Y 234.577,Z 542.236,A -85,B 0,C 180,E1 -20130.985,E2 -20130.985} C_VEL
LIN {X 0,Y 233.602,Z 550.954,A -85,B 0,C 180,E1 -20132.993,E2 -20132.993} C_VEL
LIN {X 0,Y 235.346,Z 573.727,A -85,B 0,C 180,E1 -20134.242,E2 -20134.242} C_VEL
LIN {X 0,Y 236.363,Z 584.562,A -85,B 0,C 180,E1 -20134.837,E2 -20134.837} C_VEL
LIN {X 0,Y 232.803,Z 660.64,A -85,B 0,C 180,E1 -20138.645,E2 -20138.645} C_VEL
LIN {X 0,Y 231.974,Z 675.679,A -85,B 0,C 180,E1 -20139.702,E2 -20139.702} C_VEL
LIN {X 0,Y 230.931,Z 690.052,A -85,B 0,C 180,E1 -20141.134,E2 -20141.134} C_VEL
LIN {X 0,Y 229.797,Z 701.788,A -85,B 0,C 180,E1 -20142.651,E2 -20142.651} C_VEL
LIN {X 0,Y 228.876,Z 712.663,A -85,B 0,C 180,E1 -20144.414,E2 -20144.414} C_VEL
LIN {X 0,Y 227.97,Z 722.76,A -85,B 0,C 180,E1 -20146.404,E2 -20146.404} C_VEL
LIN {X 0,Y 227.097,Z 732.82,A -85,B 0,C 180,E1 -20148.848,E2 -20148.848} C_VEL
LIN {X 0,Y 226.414,Z 741.761,A -85,B 0,C 180,E1 -20151.521,E2 -20151.521} C_VEL
LIN {X 0,Y 225.993,Z 749.277,A -85,B 0,C 180,E1 -20154.355,E2 -20154.355} C_VEL
LIN {X 0,Y 225.865,Z 755.49,A -85,B 0,C 180,E1 -20157.325,E2 -20157.325} C_VEL
LIN {X 0,Y 225.784,Z 759.714,A -85,B 0,C 180,E1 -20160,E2 -20160} C_VEL
LIN {X 0,Y 225.843,Z 761.906,A -85,B 0,C 180,E1 -20161.783,E2 -20161.783} C_VEL
LIN {X 0,Y 226.146,Z 765.035,A -85,B 0,C 180,E1 -20165.35,E2 -20165.35} C_VEL
LIN {X 0,Y 226.647,Z 765.956,A -85,B 0,C 180,E1 -20167.125,E2 -20167.125} C_VEL
LIN {X 0,Y 227.977,Z 766.595,A -85,B 0,C 180,E1 -20170.659,E2 -20170.659} C_VEL
LIN {X 0,Y 229.498,Z 766.056,A -85,B 0,C 180,E1 -20173.133,E2 -20173.133} C_VEL
LIN {X 0,Y 231.621,Z 764.606,A -85,B 0,C 180,E1 -20175.848,E2 -20175.848} C_VEL
LIN {X 0,Y 233.564,Z 762.745,A -85,B 0,C 180,E1 -20177.918,E2 -20177.918} C_VEL
LIN {X 0,Y 234.557,Z 761.334,A -85,B 0,C 180,E1 -20179.299,E2 -20179.299} C_VEL
LIN {X 0,Y 234.799,Z 758.909,A -85,B 0,C 180,E1 -20181.65,E2 -20181.65} C_VEL
LIN {X 0,Y 235.408,Z 756.025,A -85,B 0,C 180,E1 -20183.946,E2 -20183.946} C_VEL
LIN {X 0,Y 236.924,Z 753.74,A -85,B 0,C 180,E1 -20185.209,E2 -20185.209} C_VEL
LIN {X 0,Y 242.712,Z 746.427,A -85,B 0,C 180,E1 -20188.069,E2 -20188.069} C_VEL
LIN {X 0,Y 247.783,Z 739.185,A -85,B 0,C 180,E1 -20190.229,E2 -20190.229} C_VEL
LIN {X 0,Y 253.305,Z 730.499,A -85,B 0,C 180,E1 -20192.283,E2 -20192.283} C_VEL
LIN {X 0,Y 258.181,Z 721.78,A -85,B 0,C 180,E1 -20193.92,E2 -20193.92} C_VEL
LIN {X 0,Y 264,Z 710.252,A -85,B 0,C 180,E1 -20195.615,E2 -20195.615} C_VEL
LIN {X 0,Y 269.604,Z 697.205,A -85,B 0,C 180,E1 -20197.072,E2 -20197.072} C_VEL
LIN {X 0,Y 273.689,Z 685.986,A -85,B 0,C 180,E1 -20198.046,E2 -20198.046} C_VEL
LIN {X 0,Y 277.924,Z 671.647,A -85,B 0,C 180,E1 -20198.978,E2 -20198.978} C_VEL
LIN {X 0,Y 291.749,Z 611.786,A -85,B 0,C 180,E1 -20201.689,E2 -20201.689} C_VEL
LIN {X 0,Y 291.703,Z 608.928,A -85,B 0,C 180,E1 -20203.259,E2 -20203.259} C_VEL
LIN {X 0,Y 291.779,Z 607.636,A -85,B 0,C 180,E1 -20204.715,E2 -20204.715} C_VEL
LIN {X 0,Y 292.207,Z 607.253,A -85,B 0,C 180,E1 -20206.613,E2 -20206.613} C_VEL
LIN {X 0,Y 292.215,Z 607.326,A -85,B 0,C 180,E1 -20206.696,E2 -20206.696} C_VEL
LIN {X 0,Y 275.805,Z 675.915,A -85,B 0,C 180,E1 -20209.953,E2 -20209.953} C_VEL
LIN {X 0,Y 270.882,Z 691.608,A -85,B 0,C 180,E1 -20210.964,E2 -20210.964} C_VEL
LIN {X 0,Y 265.932,Z 704.462,A -85,B 0,C 180,E1 -20212.088,E2 -20212.088} C_VEL
LIN {X 0,Y 259.76,Z 718.196,A -85,B 0,C 180,E1 -20213.712,E2 -20213.712} C_VEL
LIN {X 0,Y 253.985,Z 729.324,A -85,B 0,C 180,E1 -20215.441,E2 -20215.441} C_VEL
LIN {X 0,Y 248.184,Z 739.482,A -85,B 0,C 180,E1 -20217.45,E2 -20217.45} C_VEL
LIN {X 0,Y 242.813,Z 747.95,A -85,B 0,C 180,E1 -20219.567,E2 -20219.567} C_VEL
LIN {X 0,Y 237.17,Z 756.112,A -85,B 0,C 180,E1 -20222.179,E2 -20222.179} C_VEL
LIN {X 0,Y 232.343,Z 762.653,A -85,B 0,C 180,E1 -20224.946,E2 -20224.946} C_VEL
LIN {X 0,Y 228.637,Z 767.267,A -85,B 0,C 180,E1 -20227.465,E2 -20227.465} C_VEL
LIN {X 0,Y 225.748,Z 770.714,A -85,B 0,C 180,E1 -20229.974,E2 -20229.974} C_VEL
LIN {X 0,Y 222.539,Z 774.068,A -85,B 0,C 180,E1 -20233.487,E2 -20233.487} C_VEL
LIN {X 0,Y 220.367,Z 775.921,A -85,B 0,C 180,E1 -20237.1,E2 -20237.1} C_VEL
LIN {X 0,Y 219.12,Z 776.274,A -85,B 0,C 180,E1 -20240.772,E2 -20240.772} C_VEL
LIN {X 0,Y 218.716,Z 775.037,A -85,B 0,C 180,E1 -20244.468,E2 -20244.468} C_VEL
LIN {X 0,Y 218.778,Z 773.845,A -85,B 0,C 180,E1 -20246.316,E2 -20246.316} C_VEL
LIN {X 0,Y 218.911,Z 771.158,A -85,B 0,C 180,E1 -20249.31,E2 -20249.31} C_VEL
LIN {X 0,Y 218.754,Z 773.635,A -85,B 0,C 180,E1 -20251.841,E2 -20251.841} C_VEL
LIN {X 0,Y 218.668,Z 775.59,A -85,B 0,C 180,E1 -20254.901,E2 -20254.901} C_VEL
LIN {X 0,Y 218.761,Z 776.476,A -85,B 0,C 180,E1 -20257.383,E2 -20257.383} C_VEL
LIN {X 0,Y 219.512,Z 776.671,A -85,B 0,C 180,E1 -20261.075,E2 -20261.075} C_VEL
LIN {X 0,Y 221.061,Z 775.564,A -85,B 0,C 180,E1 -20264.734,E2 -20264.734} C_VEL
LIN {X 0,Y 223.711,Z 773.18,A -85,B 0,C 180,E1 -20268.31,E2 -20268.31} C_VEL
LIN {X 0,Y 227.082,Z 769.485,A -85,B 0,C 180,E1 -20271.802,E2 -20271.802} C_VEL
LIN {X 0,Y 231.448,Z 764.429,A -85,B 0,C 180,E1 -20275.158,E2 -20275.158} C_VEL
LIN {X 0,Y 236.845,Z 757.894,A -85,B 0,C 180,E1 -20278.345,E2 -20278.345} C_VEL
LIN {X 0,Y 242.326,Z 750.764,A -85,B 0,C 180,E1 -20280.984,E2 -20280.984} C_VEL
LIN {X 0,Y 248.427,Z 742.24,A -85,B 0,C 180,E1 -20283.481,E2 -20283.481} C_VEL
LIN {X 0,Y 255.243,Z 731.861,A -85,B 0,C 180,E1 -20285.811,E2 -20285.811} C_VEL
LIN {X 0,Y 261.597,Z 721.313,A -85,B 0,C 180,E1 -20287.676,E2 -20287.676} C_VEL
LIN {X 0,Y 268.349,Z 708.695,A -85,B 0,C 180,E1 -20289.428,E2 -20289.428} C_VEL
LIN {X 0,Y 273.751,Z 697.333,A -85,B 0,C 180,E1 -20290.652,E2 -20290.652} C_VEL
LIN {X 0,Y 280.121,Z 681.812,A -85,B 0,C 180,E1 -20291.913,E2 -20291.913} C_VEL
LIN {X 0,Y 284.76,Z 668.101,A -85,B 0,C 180,E1 -20292.743,E2 -20292.743} C_VEL
LIN {X 0,Y 288.892,Z 652.446,A -85,B 0,C 180,E1 -20293.473,E2 -20293.473} C_VEL
LIN {X 0,Y 297.684,Z 615.914,A -85,B 0,C 180,E1 -20294.971,E2 -20294.971} C_VEL
LIN {X 0,Y 297.258,Z 615.946,A -85,B 0,C 180,E1 -20297.488,E2 -20297.488} C_VEL
LIN {X 0,Y 297.205,Z 617.055,A -85,B 0,C 180,E1 -20298.538,E2 -20298.538} C_VEL
LIN {X 0,Y 297.162,Z 617.523,A -85,B 0,C 180,E1 -20298.821,E2 -20298.821} C_VEL
LIN {X 0,Y 286.244,Z 661.336,A -85,B 0,C 180,E1 -20300.785,E2 -20300.785} C_VEL
LIN {X 0,Y 282.247,Z 674.003,A -85,B 0,C 180,E1 -20301.501,E2 -20301.501} C_VEL
LIN {X 0,Y 277.132,Z 687.427,A -85,B 0,C 180,E1 -20302.509,E2 -20302.509} C_VEL
LIN {X 0,Y 270.67,Z 701.715,A -85,B 0,C 180,E1 -20303.97,E2 -20303.97} C_VEL
LIN {X 0,Y 265.459,Z 711.838,A -85,B 0,C 180,E1 -20305.305,E2 -20305.305} C_VEL
LIN {X 0,Y 258.002,Z 724.609,A -85,B 0,C 180,E1 -20307.453,E2 -20307.453} C_VEL
LIN {X 0,Y 252.099,Z 733.594,A -85,B 0,C 180,E1 -20309.418,E2 -20309.418} C_VEL
LIN {X 0,Y 246.618,Z 741.254,A -85,B 0,C 180,E1 -20311.489,E2 -20311.489} C_VEL
LIN {X 0,Y 240.756,Z 748.566,A -85,B 0,C 180,E1 -20314.032,E2 -20314.032} C_VEL
LIN {X 0,Y 236.356,Z 753.68,A -85,B 0,C 180,E1 -20316.333,E2 -20316.333} C_VEL
LIN {X 0,Y 231.242,Z 758.964,A -85,B 0,C 180,E1 -20319.542,E2 -20319.542} C_VEL
LIN {X 0,Y 227.94,Z 761.879,A -85,B 0,C 180,E1 -20322.042,E2 -20322.042} C_VEL
LIN {X 0,Y 224.314,Z 764.439,A -85,B 0,C 180,E1 -20325.484,E2 -20325.484} C_VEL
LIN {X 0,Y 221.77,Z 765.497,A -85,B 0,C 180,E1 -20329.039,E2 -20329.039} C_VEL
LIN {X 0,Y 219.911,Z 765.028,A -85,B 0,C 180,E1 -20332.656,E2 -20332.656} C_VEL
LIN {X 0,Y 219.043,Z 763.047,A -85,B 0,C 180,E1 -20336.321,E2 -20336.321} C_VEL
LIN {X 0,Y 218.764,Z 760.507,A -85,B 0,C 180,E1 -20339.08,E2 -20339.08} C_VEL
LIN {X 0,Y 218.712,Z 756.992,A -85,B 0,C 180,E1 -20341.841,E2 -20341.841} C_VEL
LIN {X 0,Y 218.757,Z 751.324,A -85,B 0,C 180,E1 -20345.163,E2 -20345.163} C_VEL
LIN {X 0,Y 219.069,Z 745.467,A -85,B 0,C 180,E1 -20347.836,E2 -20347.836} C_VEL
LIN {X 0,Y 219.555,Z 737.955,A -85,B 0,C 180,E1 -20350.606,E2 -20350.606} C_VEL
LIN {X 0,Y 220.414,Z 728.698,A -85,B 0,C 180,E1 -20353.366,E2 -20353.366} C_VEL
LIN {X 0,Y 221.347,Z 718.31,A -85,B 0,C 180,E1 -20355.894,E2 -20355.894} C_VEL
LIN {X 0,Y 222.597,Z 706.822,A -85,B 0,C 180,E1 -20358.167,E2 -20358.167} C_VEL
LIN {X 0,Y 223.96,Z 694.155,A -85,B 0,C 180,E1 -20360.193,E2 -20360.193} C_VEL
LIN {X 0,Y 225.229,Z 680.775,A -85,B 0,C 180,E1 -20361.87,E2 -20361.87} C_VEL
LIN {X 0,Y 226.288,Z 667.016,A -85,B 0,C 180,E1 -20363.206,E2 -20363.206} C_VEL
LIN {X 0,Y 227.334,Z 652.232,A -85,B 0,C 180,E1 -20364.242,E2 -20364.242} C_VEL
LIN {X 0,Y 231.367,Z 582.315,A -85,B 0,C 180,E1 -20367.948,E2 -20367.948} C_VEL
LIN {X 0,Y 228.24,Z 550.155,A -85,B 0,C 180,E1 -20369.909,E2 -20369.909} C_VEL
LIN {X 0,Y 227.301,Z 537.926,A -85,B 0,C 180,E1 -20370.673,E2 -20370.673} C_VEL
LIN {X 0,Y 224.863,Z 526.247,A -85,B 0,C 180,E1 -20374.829,E2 -20374.829} C_VEL
LIN {X 0,Y 222.25,Z 514.537,A -85,B 0,C 180,E1 -20379.23,E2 -20379.23} C_VEL
LIN {X 0,Y 220.813,Z 508.103,A -85,B 0,C 180,E1 -20381.77,E2 -20381.77} C_VEL
LIN {X 0,Y 220.775,Z 508.111,A -85,B 0,C 180,E1 -20385.546,E2 -20385.546} C_VEL
LIN {X 0,Y 220.808,Z 508.104,A -85,B 0,C 180,E1 -20390.463,E2 -20390.463} C_VEL
LIN {X 0,Y 220.805,Z 508.103,A -85,B 0,C 180,E1 -20395.045,E2 -20395.045} C_VEL
LIN {X 0,Y 220.869,Z 508.098,A -85,B 0,C 180,E1 -20399.395,E2 -20399.395} C_VEL
LIN {X 0,Y 220.897,Z 508.092,A -85,B 0,C 180,E1 -20403.549,E2 -20403.549} C_VEL
LIN {X 0,Y 220.88,Z 508.098,A -85,B 0,C 180,E1 -20407.553,E2 -20407.553} C_VEL
LIN {X 0,Y 220.986,Z 508.078,A -85,B 0,C 180,E1 -20412.571,E2 -20412.571} C_VEL
LIN {X 0,Y 221.028,Z 508.078,A -85,B 0,C 180,E1 -20417.139,E2 -20417.139} C_VEL
LIN {X 0,Y 221.259,Z 508.045,A -85,B 0,C 180,E1 -20420.862,E2 -20420.862} C_VEL
LIN {X 0,Y 221.313,Z 508.039,A -85,B 0,C 180,E1 -20422.702,E2 -20422.702} C_VEL
LIN {X 0,Y 221.517,Z 508.013,A -85,B 0,C 180,E1 -20428.182,E2 -20428.182} C_VEL
LIN {X 0,Y 221.515,Z 508.016,A -85,B 0,C 180,E1 -20431.818,E2 -20431.818} C_VEL
LIN {X 0,Y 221.313,Z 508.042,A -85,B 0,C 180,E1 -20437.298,E2 -20437.298} C_VEL
LIN {X 0,Y 221.118,Z 508.065,A -85,B 0,C 180,E1 -20440.994,E2 -20440.994} C_VEL
LIN {X 0,Y 221.018,Z 508.074,A -85,B 0,C 180,E1 -20446.63,E2 -20446.63} C_VEL
LIN {X 0,Y 220.894,Z 508.092,A -85,B 0,C 180,E1 -20450.486,E2 -20450.486} C_VEL
LIN {X 0,Y 220.868,Z 508.093,A -85,B 0,C 180,E1 -20454.435,E2 -20454.435} C_VEL
LIN {X 0,Y 220.828,Z 508.101,A -85,B 0,C 180,E1 -20458.515,E2 -20458.515} C_VEL
LIN {X 0,Y 220.824,Z 508.1,A -85,B 0,C 180,E1 -20462.755,E2 -20462.755} C_VEL
LIN {X 0,Y 220.839,Z 508.103,A -85,B 0,C 180,E1 -20467.288,E2 -20467.288} C_VEL
LIN {X 0,Y 220.777,Z 508.104,A -85,B 0,C 180,E1 -20471.951,E2 -20471.951} C_VEL
LIN {X 0,Y 220.777,Z 508.11,A -85,B 0,C 180,E1 -20475.547,E2 -20475.547} C_VEL
LIN {X 0,Y 220.809,Z 508.105,A -85,B 0,C 180,E1 -20480.464,E2 -20480.464} C_VEL
LIN {X 0,Y 220.873,Z 508.293,A -85,B 0,C 180,E1 -20481.607,E2 -20481.607} C_VEL
LIN {X 0,Y 224.325,Z 523.264,A -85,B 0,C 180,E1 -20485.672,E2 -20485.672} C_VEL
LIN {X 0,Y 227.784,Z 538.866,A -85,B 0,C 180,E1 -20489.758,E2 -20489.758} C_VEL
LIN {X 0,Y 227.763,Z 541.587,A -85,B 0,C 180,E1 -20490.416,E2 -20490.416} C_VEL
LIN {X 0,Y 226.648,Z 551.341,A -85,B 0,C 180,E1 -20492.664,E2 -20492.664} C_VEL
LIN {X 0,Y 228.276,Z 573.779,A -85,B 0,C 180,E1 -20493.94,E2 -20493.94} C_VEL
LIN {X 0,Y 229.361,Z 584.394,A -85,B 0,C 180,E1 -20494.548,E2 -20494.548} C_VEL
LIN {X 0,Y 225.727,Z 660.703,A -85,B 0,C 180,E1 -20498.523,E2 -20498.523} C_VEL
LIN {X 0,Y 224.933,Z 675.115,A -85,B 0,C 180,E1 -20499.576,E2 -20499.576} C_VEL
LIN {X 0,Y 223.991,Z 687.753,A -85,B 0,C 180,E1 -20500.844,E2 -20500.844} C_VEL
LIN {X 0,Y 222.942,Z 699.387,A -85,B 0,C 180,E1 -20502.337,E2 -20502.337} C_VEL
LIN {X 0,Y 221.981,Z 710.775,A -85,B 0,C 180,E1 -20504.153,E2 -20504.153} C_VEL
LIN {X 0,Y 221.009,Z 721.175,A -85,B 0,C 180,E1 -20506.202,E2 -20506.202} C_VEL
LIN {X 0,Y 220.165,Z 730.775,A -85,B 0,C 180,E1 -20508.492,E2 -20508.492} C_VEL
LIN {X 0,Y 219.441,Z 740.119,A -85,B 0,C 180,E1 -20511.25,E2 -20511.25} C_VEL
LIN {X 0,Y 219.083,Z 746.477,A -85,B 0,C 180,E1 -20513.554,E2 -20513.554} C_VEL
LIN {X 0,Y 218.846,Z 752.699,A -85,B 0,C 180,E1 -20516.318,E2 -20516.318} C_VEL
LIN {X 0,Y 218.71,Z 757.62,A -85,B 0,C 180,E1 -20519.079,E2 -20519.079} C_VEL
LIN {X 0,Y 218.78,Z 761.395,A -85,B 0,C 180,E1 -20521.841,E2 -20521.841} C_VEL
LIN {X 0,Y 218.834,Z 763.315,A -85,B 0,C 180,E1 -20523.683,E2 -20523.683} C_VEL
LIN {X 0,Y 219.598,Z 765.88,A -85,B 0,C 180,E1 -20527.355,E2 -20527.355} C_VEL
LIN {X 0,Y 220.23,Z 766.589,A -85,B 0,C 180,E1 -20529.181,E2 -20529.181} C_VEL
LIN {X 0,Y 221.024,Z 766.883,A -85,B 0,C 180,E1 -20530.999,E2 -20530.999} C_VEL
LIN {X 0,Y 223.396,Z 766.28,A -85,B 0,C 180,E1 -20534.577,E2 -20534.577} C_VEL
LIN {X 0,Y 226.463,Z 764.179,A -85,B 0,C 180,E1 -20538.08,E2 -20538.08} C_VEL
LIN {X 0,Y 230.751,Z 760.402,A -85,B 0,C 180,E1 -20541.437,E2 -20541.437} C_VEL
LIN {X 0,Y 234.536,Z 756.46,A -85,B 0,C 180,E1 -20543.862,E2 -20543.862} C_VEL
LIN {X 0,Y 236.924,Z 753.74,A -85,B 0,C 180,E1 -20545.209,E2 -20545.209} C_VEL
LIN {X 0,Y 238.594,Z 751.309,A -85,B 0,C 180,E1 -20546.446,E2 -20546.446} C_VEL
LIN {X 0,Y 240.097,Z 747.438,A -85,B 0,C 180,E1 -20548.606,E2 -20548.606} C_VEL
LIN {X 0,Y 241.878,Z 743.038,A -85,B 0,C 180,E1 -20550.659,E2 -20550.659} C_VEL
LIN {X 0,Y 243.905,Z 739.795,A -85,B 0,C 180,E1 -20551.707,E2 -20551.707} C_VEL
LIN {X 0,Y 249.807,Z 731.17,A -85,B 0,C 180,E1 -20553.755,E2 -20553.755} C_VEL
LIN {X 0,Y 254.987,Z 722.638,A -85,B 0,C 180,E1 -20555.367,E2 -20555.367} C_VEL
LIN {X 0,Y 261.13,Z 711.314,A -85,B 0,C 180,E1 -20557.027,E2 -20557.027} C_VEL
LIN {X 0,Y 266.387,Z 700.001,A -85,B 0,C 180,E1 -20558.316,E2 -20558.316} C_VEL
LIN {X 0,Y 271.282,Z 687.749,A -85,B 0,C 180,E1 -20559.399,E2 -20559.399} C_VEL
LIN {X 0,Y 275.382,Z 675.114,A -85,B 0,C 180,E1 -20560.241,E2 -20560.241} C_VEL
LIN {X 0,Y 280.254,Z 655.835,A -85,B 0,C 180,E1 -20561.174,E2 -20561.174} C_VEL
LIN {X 0,Y 289.78,Z 616.644,A -85,B 0,C 180,E1 -20562.917,E2 -20562.917} C_VEL
LIN {X 0,Y 289.854,Z 615.061,A -85,B 0,C 180,E1 -20564.057,E2 -20564.057} C_VEL
LIN {X 0,Y 290.012,Z 614.241,A -85,B 0,C 180,E1 -20565.35,E2 -20565.35} C_VEL
LIN {X 0,Y 290.035,Z 614.349,A -85,B 0,C 180,E1 -20565.585,E2 -20565.585} C_VEL
LIN {X 0,Y 274.549,Z 675.556,A -85,B 0,C 180,E1 -20568.459,E2 -20568.459} C_VEL
LIN {X 0,Y 269.739,Z 690.171,A -85,B 0,C 180,E1 -20569.355,E2 -20569.355} C_VEL
LIN {X 0,Y 264.62,Z 702.803,A -85,B 0,C 180,E1 -20570.401,E2 -20570.401} C_VEL
LIN {X 0,Y 259.18,Z 714.4,A -85,B 0,C 180,E1 -20571.663,E2 -20571.663} C_VEL
LIN {X 0,Y 252.919,Z 726.05,A -85,B 0,C 180,E1 -20573.314,E2 -20573.314} C_VEL
LIN {X 0,Y 247.59,Z 735.001,A -85,B 0,C 180,E1 -20574.914,E2 -20574.914} C_VEL
LIN {X 0,Y 240.649,Z 745.417,A -85,B 0,C 180,E1 -20577.297,E2 -20577.297} C_VEL
LIN {X 0,Y 234.371,Z 753.909,A -85,B 0,C 180,E1 -20579.849,E2 -20579.849} C_VEL
LIN {X 0,Y 228.891,Z 760.751,A -85,B 0,C 180,E1 -20582.576,E2 -20582.576} C_VEL
LIN {X 0,Y 224.153,Z 766.178,A -85,B 0,C 180,E1 -20585.402,E2 -20585.402} C_VEL
LIN {X 0,Y 220.11,Z 770.442,A -85,B 0,C 180,E1 -20588.458,E2 -20588.458} C_VEL
LIN {X 0,Y 217.311,Z 773.063,A -85,B 0,C 180,E1 -20591.131,E2 -20591.131} C_VEL
LIN {X 0,Y 214.406,Z 775.3,A -85,B 0,C 180,E1 -20594.798,E2 -20594.798} C_VEL
LIN {X 0,Y 212.655,Z 776.026,A -85,B 0,C 180,E1 -20598.563,E2 -20598.563} C_VEL
LIN {X 0,Y 211.769,Z 775.283,A -85,B 0,C 180,E1 -20602.372,E2 -20602.372} C_VEL
LIN {X 0,Y 211.687,Z 773.939,A -85,B 0,C 180,E1 -20604.872,E2 -20604.872} C_VEL
LIN {X 0,Y 211.823,Z 771.141,A -85,B 0,C 180,E1 -20608.099,E2 -20608.099} C_VEL
LIN {X 0,Y 211.948,Z 769.96,A -85,B 0,C 180,E1 -20609.169,E2 -20609.169} C_VEL
LIN {X 0,Y 211.728,Z 772.686,A -85,B 0,C 180,E1 -20611.902,E2 -20611.902} C_VEL
LIN {X 0,Y 211.617,Z 774.795,A -85,B 0,C 180,E1 -20614.91,E2 -20614.91} C_VEL
LIN {X 0,Y 211.714,Z 775.935,A -85,B 0,C 180,E1 -20617.631,E2 -20617.631} C_VEL
LIN {X 0,Y 212.505,Z 776.409,A -85,B 0,C 180,E1 -20621.446,E2 -20621.446} C_VEL
LIN {X 0,Y 214.189,Z 775.601,A -85,B 0,C 180,E1 -20625.218,E2 -20625.218} C_VEL
LIN {X 0,Y 216.953,Z 773.526,A -85,B 0,C 180,E1 -20628.902,E2 -20628.902} C_VEL
LIN {X 0,Y 220.535,Z 770.2,A -85,B 0,C 180,E1 -20632.484,E2 -20632.484} C_VEL
LIN {X 0,Y 225.129,Z 765.533,A -85,B 0,C 180,E1 -20635.916,E2 -20635.916} C_VEL
LIN {X 0,Y 230.772,Z 759.395,A -85,B 0,C 180,E1 -20639.161,E2 -20639.161} C_VEL
LIN {X 0,Y 237.352,Z 751.711,A -85,B 0,C 180,E1 -20642.207,E2 -20642.207} C_VEL
LIN {X 0,Y 243.792,Z 743.476,A -85,B 0,C 180,E1 -20644.705,E2 -20644.705} C_VEL
LIN {X 0,Y 250.952,Z 733.622,A -85,B 0,C 180,E1 -20647.022,E2 -20647.022} C_VEL
LIN {X 0,Y 258.706,Z 721.667,A -85,B 0,C 180,E1 -20649.169,E2 -20649.169} C_VEL
LIN {X 0,Y 265.195,Z 710.414,A -85,B 0,C 180,E1 -20650.738,E2 -20650.738} C_VEL
LIN {X 0,Y 271.45,Z 698.312,A -85,B 0,C 180,E1 -20652.061,E2 -20652.061} C_VEL
LIN {X 0,Y 277.411,Z 684.842,A -85,B 0,C 180,E1 -20653.159,E2 -20653.159} C_VEL
LIN {X 0,Y 282.572,Z 671.171,A -85,B 0,C 180,E1 -20654.016,E2 -20654.016} C_VEL
LIN {X 0,Y 287.409,Z 654.773,A -85,B 0,C 180,E1 -20654.797,E2 -20654.797} C_VEL
LIN {X 0,Y 295.546,Z 622.615,A -85,B 0,C 180,E1 -20656.113,E2 -20656.113} C_VEL
LIN {X 0,Y 295.417,Z 622.886,A -85,B 0,C 180,E1 -20657.585,E2 -20657.585} C_VEL
LIN {X 0,Y 295.252,Z 623.564,A -85,B 0,C 180,E1 -20657.673,E2 -20657.673} C_VEL
LIN {X 0,Y 284.579,Z 663.877,A -85,B 0,C 180,E1 -20659.472,E2 -20659.472} C_VEL
LIN {X 0,Y 280.77,Z 675.059,A -85,B 0,C 180,E1 -20660.102,E2 -20660.102} C_VEL
LIN {X 0,Y 275.422,Z 688.086,A -85,B 0,C 180,E1 -20661.071,E2 -20661.071} C_VEL
LIN {X 0,Y 269.125,Z 701.302,A -85,B 0,C 180,E1 -20662.38,E2 -20662.38} C_VEL
LIN {X 0,Y 263.559,Z 711.384,A -85,B 0,C 180,E1 -20663.655,E2 -20663.655} C_VEL
LIN {X 0,Y 256.848,Z 722.398,A -85,B 0,C 180,E1 -20665.422,E2 -20665.422} C_VEL
LIN {X 0,Y 249.414,Z 733.109,A -85,B 0,C 180,E1 -20667.63,E2 -20667.63} C_VEL
LIN {X 0,Y 242.596,Z 741.897,A -85,B 0,C 180,E1 -20670.018,E2 -20670.018} C_VEL
LIN {X 0,Y 236.323,Z 749.133,A -85,B 0,C 180,E1 -20672.551,E2 -20672.551} C_VEL
LIN {X 0,Y 230.093,Z 755.61,A -85,B 0,C 180,E1 -20675.648,E2 -20675.648} C_VEL
LIN {X 0,Y 226,Z 759.349,A -85,B 0,C 180,E1 -20678.089,E2 -20678.089} C_VEL
LIN {X 0,Y 221.298,Z 763.023,A -85,B 0,C 180,E1 -20681.483,E2 -20681.483} C_VEL
LIN {X 0,Y 217.501,Z 765.153,A -85,B 0,C 180,E1 -20685.019,E2 -20685.019} C_VEL
LIN {X 0,Y 214.823,Z 765.831,A -85,B 0,C 180,E1 -20688.68,E2 -20688.68} C_VEL
LIN {X 0,Y 212.883,Z 765.055,A -85,B 0,C 180,E1 -20692.412,E2 -20692.412} C_VEL
LIN {X 0,Y 211.975,Z 762.746,A -85,B 0,C 180,E1 -20696.198,E2 -20696.198} C_VEL
LIN {X 0,Y 211.702,Z 759.985,A -85,B 0,C 180,E1 -20699.049,E2 -20699.049} C_VEL
LIN {X 0,Y 211.65,Z 756.211,A -85,B 0,C 180,E1 -20701.903,E2 -20701.903} C_VEL
LIN {X 0,Y 211.72,Z 750.424,A -85,B 0,C 180,E1 -20705.221,E2 -20705.221} C_VEL
LIN {X 0,Y 212.066,Z 744.032,A -85,B 0,C 180,E1 -20708.097,E2 -20708.097} C_VEL
LIN {X 0,Y 212.598,Z 736.192,A -85,B 0,C 180,E1 -20710.958,E2 -20710.958} C_VEL
LIN {X 0,Y 213.51,Z 726.55,A -85,B 0,C 180,E1 -20713.807,E2 -20713.807} C_VEL
LIN {X 0,Y 214.472,Z 715.564,A -85,B 0,C 180,E1 -20716.417,E2 -20716.417} C_VEL
LIN {X 0,Y 215.879,Z 703.496,A -85,B 0,C 180,E1 -20718.753,E2 -20718.753} C_VEL
LIN {X 0,Y 217.31,Z 689.896,A -85,B 0,C 180,E1 -20720.839,E2 -20720.839} C_VEL
LIN {X 0,Y 218.452,Z 676.474,A -85,B 0,C 180,E1 -20722.46,E2 -20722.46} C_VEL
LIN {X 0,Y 219.673,Z 661.565,A -85,B 0,C 180,E1 -20723.823,E2 -20723.823} C_VEL
LIN {X 0,Y 220.846,Z 642.876,A -85,B 0,C 180,E1 -20725.002,E2 -20725.002} C_VEL
LIN {X 0,Y 224.387,Z 582.96,A -85,B 0,C 180,E1 -20728.28,E2 -20728.28} C_VEL
LIN {X 0,Y 221.309,Z 550.083,A -85,B 0,C 180,E1 -20730.36,E2 -20730.36} C_VEL
LIN {X 0,Y 220.605,Z 539.931,A -85,B 0,C 180,E1 -20730.991,E2 -20730.991} C_VEL
LIN {X 0,Y 220.021,Z 537.747,A -85,B 0,C 180,E1 -20731.202,E2 -20731.202} C_VEL
LIN {X 0,Y 217.519,Z 525.92,A -85,B 0,C 180,E1 -20735.562,E2 -20735.562} C_VEL
LIN {X 0,Y 215.061,Z 514.919,A -85,B 0,C 180,E1 -20739.83,E2 -20739.83} C_VEL
LIN {X 0,Y 213.751,Z 508.982,A -85,B 0,C 180,E1 -20742.286,E2 -20742.286} C_VEL
LIN {X 0,Y 213.707,Z 508.989,A -85,B 0,C 180,E1 -20746.344,E2 -20746.344} C_VEL
LIN {X 0,Y 213.718,Z 508.989,A -85,B 0,C 180,E1 -20749.143,E2 -20749.143} C_VEL
LIN {X 0,Y 213.746,Z 508.984,A -85,B 0,C 180,E1 -20753.712,E2 -20753.712} C_VEL
LIN {X 0,Y 213.797,Z 508.976,A -85,B 0,C 180,E1 -20758.724,E2 -20758.724} C_VEL
LIN {X 0,Y 213.827,Z 508.971,A -85,B 0,C 180,E1 -20762.603,E2 -20762.603} C_VEL
LIN {X 0,Y 213.854,Z 508.97,A -85,B 0,C 180,E1 -20766.953,E2 -20766.953} C_VEL
LIN {X 0,Y 213.945,Z 508.955,A -85,B 0,C 180,E1 -20772.804,E2 -20772.804} C_VEL
LIN {X 0,Y 213.982,Z 508.954,A -85,B 0,C 180,E1 -20776.708,E2 -20776.708} C_VEL
LIN {X 0,Y 214.198,Z 508.924,A -85,B 0,C 180,E1 -20780.558,E2 -20780.558} C_VEL
LIN {X 0,Y 214.25,Z 508.918,A -85,B 0,C 180,E1 -20782.46,E2 -20782.46} C_VEL
LIN {X 0,Y 214.45,Z 508.894,A -85,B 0,C 180,E1 -20788.122,E2 -20788.122} C_VEL
LIN {X 0,Y 214.556,Z 508.88,A -85,B 0,C 180,E1 -20790,E2 -20790} C_VEL
LIN {X 0,Y 214.448,Z 508.896,A -85,B 0,C 180,E1 -20791.878,E2 -20791.878} C_VEL
LIN {X 0,Y 214.25,Z 508.919,A -85,B 0,C 180,E1 -20797.54,E2 -20797.54} C_VEL
LIN {X 0,Y 214.049,Z 508.948,A -85,B 0,C 180,E1 -20801.362,E2 -20801.362} C_VEL
LIN {X 0,Y 213.936,Z 508.961,A -85,B 0,C 180,E1 -20805.237,E2 -20805.237} C_VEL
LIN {X 0,Y 213.87,Z 508.969,A -85,B 0,C 180,E1 -20809.184,E2 -20809.184} C_VEL
LIN {X 0,Y 213.848,Z 508.973,A -85,B 0,C 180,E1 -20813.227,E2 -20813.227} C_VEL
LIN {X 0,Y 213.83,Z 508.975,A -85,B 0,C 180,E1 -20817.45,E2 -20817.45} C_VEL
LIN {X 0,Y 213.771,Z 508.98,A -85,B 0,C 180,E1 -20821.737,E2 -20821.737} C_VEL
LIN {X 0,Y 213.754,Z 508.981,A -85,B 0,C 180,E1 -20826.286,E2 -20826.286} C_VEL
LIN {X 0,Y 213.719,Z 508.988,A -85,B 0,C 180,E1 -20831.124,E2 -20831.124} C_VEL
LIN {X 0,Y 213.71,Z 508.988,A -85,B 0,C 180,E1 -20833.678,E2 -20833.678} C_VEL
LIN {X 0,Y 213.708,Z 508.988,A -85,B 0,C 180,E1 -20836.344,E2 -20836.344} C_VEL
LIN {X 0,Y 213.807,Z 509.131,A -85,B 0,C 180,E1 -20841.183,E2 -20841.183} C_VEL
LIN {X 0,Y 217.187,Z 523.584,A -85,B 0,C 180,E1 -20845.197,E2 -20845.197} C_VEL
LIN {X 0,Y 220.838,Z 540.256,A -85,B 0,C 180,E1 -20849.653,E2 -20849.653} C_VEL
LIN {X 0,Y 219.684,Z 551.46,A -85,B 0,C 180,E1 -20852.324,E2 -20852.324} C_VEL
LIN {X 0,Y 221.285,Z 574.439,A -85,B 0,C 180,E1 -20853.663,E2 -20853.663} C_VEL
LIN {X 0,Y 222.355,Z 585.308,A -85,B 0,C 180,E1 -20854.303,E2 -20854.303} C_VEL
LIN {X 0,Y 218.645,Z 660.574,A -85,B 0,C 180,E1 -20858.431,E2 -20858.431} C_VEL
LIN {X 0,Y 217.817,Z 675.31,A -85,B 0,C 180,E1 -20859.542,E2 -20859.542} C_VEL
LIN {X 0,Y 216.867,Z 688.265,A -85,B 0,C 180,E1 -20860.891,E2 -20860.891} C_VEL
LIN {X 0,Y 215.746,Z 700.044,A -85,B 0,C 180,E1 -20862.463,E2 -20862.463} C_VEL
LIN {X 0,Y 214.77,Z 711.321,A -85,B 0,C 180,E1 -20864.338,E2 -20864.338} C_VEL
LIN {X 0,Y 213.927,Z 720.634,A -85,B 0,C 180,E1 -20866.221,E2 -20866.221} C_VEL
LIN {X 0,Y 213.096,Z 730.266,A -85,B 0,C 180,E1 -20868.587,E2 -20868.587} C_VEL
LIN {X 0,Y 212.494,Z 738.283,A -85,B 0,C 180,E1 -20870.961,E2 -20870.961} C_VEL
LIN {X 0,Y 212.057,Z 745.207,A -85,B 0,C 180,E1 -20873.434,E2 -20873.434} C_VEL
LIN {X 0,Y 211.795,Z 751.522,A -85,B 0,C 180,E1 -20876.195,E2 -20876.195} C_VEL
LIN {X 0,Y 211.655,Z 756.737,A -85,B 0,C 180,E1 -20879.049,E2 -20879.049} C_VEL
LIN {X 0,Y 211.719,Z 760.734,A -85,B 0,C 180,E1 -20881.902,E2 -20881.902} C_VEL
LIN {X 0,Y 212.02,Z 764.498,A -85,B 0,C 180,E1 -20885.707,E2 -20885.707} C_VEL
LIN {X 0,Y 212.563,Z 765.759,A -85,B 0,C 180,E1 -20887.6,E2 -20887.6} C_VEL
LIN {X 0,Y 214.051,Z 767.061,A -85,B 0,C 180,E1 -20891.362,E2 -20891.362} C_VEL
LIN {X 0,Y 216.563,Z 766.858,A -85,B 0,C 180,E1 -20895.048,E2 -20895.048} C_VEL
LIN {X 0,Y 219.806,Z 765.107,A -85,B 0,C 180,E1 -20898.647,E2 -20898.647} C_VEL
LIN {X 0,Y 224.288,Z 761.804,A -85,B 0,C 180,E1 -20902.087,E2 -20902.087} C_VEL
LIN {X 0,Y 228.246,Z 758.209,A -85,B 0,C 180,E1 -20904.562,E2 -20904.562} C_VEL
LIN {X 0,Y 232.717,Z 753.627,A -85,B 0,C 180,E1 -20906.936,E2 -20906.936} C_VEL
LIN {X 0,Y 238.48,Z 746.864,A -85,B 0,C 180,E1 -20909.579,E2 -20909.579} C_VEL
LIN {X 0,Y 243.905,Z 739.795,A -85,B 0,C 180,E1 -20911.707,E2 -20911.707} C_VEL
LIN {X 0,Y 246.059,Z 736.425,A -85,B 0,C 180,E1 -20912.726,E2 -20912.726} C_VEL
LIN {X 0,Y 250.512,Z 726.814,A -85,B 0,C 180,E1 -20916.031,E2 -20916.031} C_VEL
LIN {X 0,Y 252.509,Z 722.993,A -85,B 0,C 180,E1 -20916.933,E2 -20916.933} C_VEL
LIN {X 0,Y 253.326,Z 721.58,A -85,B 0,C 180,E1 -20917.178,E2 -20917.178} C_VEL
LIN {X 0,Y 259.698,Z 710.411,A -85,B 0,C 180,E1 -20918.742,E2 -20918.742} C_VEL
LIN {X 0,Y 265.253,Z 698.903,A -85,B 0,C 180,E1 -20919.98,E2 -20919.98} C_VEL
LIN {X 0,Y 269.743,Z 688.208,A -85,B 0,C 180,E1 -20920.891,E2 -20920.891} C_VEL
LIN {X 0,Y 274.375,Z 674.662,A -85,B 0,C 180,E1 -20921.758,E2 -20921.758} C_VEL
LIN {X 0,Y 281.297,Z 648.094,A -85,B 0,C 180,E1 -20922.977,E2 -20922.977} C_VEL
LIN {X 0,Y 288.01,Z 621.968,A -85,B 0,C 180,E1 -20924.11,E2 -20924.11} C_VEL
LIN {X 0,Y 288.061,Z 621.665,A -85,B 0,C 180,E1 -20924.463,E2 -20924.463} C_VEL
LIN {X 0,Y 273.913,Z 674.669,A -85,B 0,C 180,E1 -20926.91,E2 -20926.91} C_VEL
LIN {X 0,Y 269.038,Z 688.917,A -85,B 0,C 180,E1 -20927.742,E2 -20927.742} C_VEL
LIN {X 0,Y 263.648,Z 701.536,A -85,B 0,C 180,E1 -20928.719,E2 -20928.719} C_VEL
LIN {X 0,Y 257.883,Z 713.241,A -85,B 0,C 180,E1 -20929.921,E2 -20929.921} C_VEL
LIN {X 0,Y 251.628,Z 724.213,A -85,B 0,C 180,E1 -20931.401,E2 -20931.401} C_VEL
LIN {X 0,Y 245.486,Z 733.889,A -85,B 0,C 180,E1 -20933.044,E2 -20933.044} C_VEL
LIN {X 0,Y 238.031,Z 744.353,A -85,B 0,C 180,E1 -20935.364,E2 -20935.364} C_VEL
LIN {X 0,Y 231.249,Z 752.92,A -85,B 0,C 180,E1 -20937.869,E2 -20937.869} C_VEL
LIN {X 0,Y 225.959,Z 758.954,A -85,B 0,C 180,E1 -20940.155,E2 -20940.155} C_VEL
LIN {X 0,Y 219.813,Z 765.392,A -85,B 0,C 180,E1 -20943.409,E2 -20943.409} C_VEL
LIN {X 0,Y 214.648,Z 770.224,A -85,B 0,C 180,E1 -20946.865,E2 -20946.865} C_VEL
LIN {X 0,Y 210.629,Z 773.473,A -85,B 0,C 180,E1 -20950.508,E2 -20950.508} C_VEL
LIN {X 0,Y 207.546,Z 775.309,A -85,B 0,C 180,E1 -20954.282,E2 -20954.282} C_VEL
LIN {X 0,Y 205.68,Z 775.717,A -85,B 0,C 180,E1 -20958.17,E2 -20958.17} C_VEL
LIN {X 0,Y 204.755,Z 774.603,A -85,B 0,C 180,E1 -20962.109,E2 -20962.109} C_VEL
LIN {X 0,Y 204.718,Z 771.99,A -85,B 0,C 180,E1 -20966.063,E2 -20966.063} C_VEL
LIN {X 0,Y 204.955,Z 768.734,A -85,B 0,C 180,E1 -20969.141,E2 -20969.141} C_VEL
LIN {X 0,Y 204.723,Z 771.704,A -85,B 0,C 180,E1 -20971.967,E2 -20971.967} C_VEL
LIN {X 0,Y 204.593,Z 773.96,A -85,B 0,C 180,E1 -20975.007,E2 -20975.007} C_VEL
LIN {X 0,Y 204.668,Z 775.325,A -85,B 0,C 180,E1 -20977.895,E2 -20977.895} C_VEL
LIN {X 0,Y 205.512,Z 776.067,A -85,B 0,C 180,E1 -20981.841,E2 -20981.841} C_VEL
LIN {X 0,Y 207.338,Z 775.551,A -85,B 0,C 180,E1 -20985.734,E2 -20985.734} C_VEL
LIN {X 0,Y 210.217,Z 773.805,A -85,B 0,C 180,E1 -20989.531,E2 -20989.531} C_VEL
LIN {X 0,Y 214.013,Z 770.806,A -85,B 0,C 180,E1 -20993.208,E2 -20993.208} C_VEL
LIN {X 0,Y 218.829,Z 766.543,A -85,B 0,C 180,E1 -20996.72,E2 -20996.72} C_VEL
LIN {X 0,Y 224.737,Z 760.896,A -85,B 0,C 180,E1 -21000.024,E2 -21000.024} C_VEL
LIN {X 0,Y 231.601,Z 753.714,A -85,B 0,C 180,E1 -21003.108,E2 -21003.108} C_VEL
LIN {X 0,Y 238.278,Z 746.111,A -85,B 0,C 180,E1 -21005.629,E2 -21005.629} C_VEL
LIN {X 0,Y 246.781,Z 735.415,A -85,B 0,C 180,E1 -21008.273,E2 -21008.273} C_VEL
LIN {X 0,Y 253.659,Z 725.794,A -85,B 0,C 180,E1 -21010.104,E2 -21010.104} C_VEL
LIN {X 0,Y 260.943,Z 714.566,A -85,B 0,C 180,E1 -21011.805,E2 -21011.805} C_VEL
LIN {X 0,Y 267.374,Z 703.253,A -85,B 0,C 180,E1 -21013.112,E2 -21013.112} C_VEL
LIN {X 0,Y 274.2,Z 689.702,A -85,B 0,C 180,E1 -21014.303,E2 -21014.303} C_VEL
LIN {X 0,Y 279.811,Z 676.369,A -85,B 0,C 180,E1 -21015.199,E2 -21015.199} C_VEL
LIN {X 0,Y 285.229,Z 660.627,A -85,B 0,C 180,E1 -21015.983,E2 -21015.983} C_VEL
LIN {X 0,Y 290.982,Z 639.258,A -85,B 0,C 180,E1 -21016.832,E2 -21016.832} C_VEL
LIN {X 0,Y 290.977,Z 639.227,A -85,B 0,C 180,E1 -21016.934,E2 -21016.934} C_VEL
LIN {X 0,Y 283.874,Z 664.61,A -85,B 0,C 180,E1 -21018.052,E2 -21018.052} C_VEL
LIN {X 0,Y 279.535,Z 676.491,A -85,B 0,C 180,E1 -21018.702,E2 -21018.702} C_VEL
LIN {X 0,Y 273.295,Z 690.642,A -85,B 0,C 180,E1 -21019.751,E2 -21019.751} C_VEL
LIN {X 0,Y 266.725,Z 703.298,A -85,B 0,C 180,E1 -21021.017,E2 -21021.017} C_VEL
LIN {X 0,Y 259.835,Z 714.792,A -85,B 0,C 180,E1 -21022.513,E2 -21022.513} C_VEL
LIN {X 0,Y 252.745,Z 725.232,A -85,B 0,C 180,E1 -21024.272,E2 -21024.272} C_VEL
LIN {X 0,Y 246.05,Z 734.16,A -85,B 0,C 180,E1 -21026.152,E2 -21026.152} C_VEL
LIN {X 0,Y 237.817,Z 743.827,A -85,B 0,C 180,E1 -21028.858,E2 -21028.858} C_VEL
LIN {X 0,Y 232.121,Z 749.763,A -85,B 0,C 180,E1 -21031.024,E2 -21031.024} C_VEL
LIN {X 0,Y 226.985,Z 754.697,A -85,B 0,C 180,E1 -21033.323,E2 -21033.323} C_VEL
LIN {X 0,Y 220.955,Z 759.79,A -85,B 0,C 180,E1 -21036.572,E2 -21036.572} C_VEL
LIN {X 0,Y 217.017,Z 762.62,A -85,B 0,C 180,E1 -21039.131,E2 -21039.131} C_VEL
LIN {X 0,Y 212.511,Z 765.108,A -85,B 0,C 180,E1 -21042.684,E2 -21042.684} C_VEL
LIN {X 0,Y 210.679,Z 765.817,A -85,B 0,C 180,E1 -21044.522,E2 -21044.522} C_VEL
LIN {X 0,Y 207.886,Z 766.134,A -85,B 0,C 180,E1 -21048.297,E2 -21048.297} C_VEL
LIN {X 0,Y 205.871,Z 764.97,A -85,B 0,C 180,E1 -21052.152,E2 -21052.152} C_VEL
LIN {X 0,Y 204.91,Z 762.337,A -85,B 0,C 180,E1 -21056.067,E2 -21056.067} C_VEL
LIN {X 0,Y 204.641,Z 759.303,A -85,B 0,C 180,E1 -21059.016,E2 -21059.016} C_VEL
LIN {X 0,Y 204.59,Z 755.288,A -85,B 0,C 180,E1 -21061.969,E2 -21061.969} C_VEL
LIN {X 0,Y 204.671,Z 749.492,A -85,B 0,C 180,E1 -21065.248,E2 -21065.248} C_VEL
LIN {X 0,Y 205.078,Z 742.462,A -85,B 0,C 180,E1 -21068.375,E2 -21068.375} C_VEL
LIN {X 0,Y 205.65,Z 734.233,A -85,B 0,C 180,E1 -21071.333,E2 -21071.333} C_VEL
LIN {X 0,Y 206.602,Z 724.107,A -85,B 0,C 180,E1 -21074.278,E2 -21074.278} C_VEL
LIN {X 0,Y 207.525,Z 713.837,A -85,B 0,C 180,E1 -21076.73,E2 -21076.73} C_VEL
LIN {X 0,Y 208.845,Z 702.673,A -85,B 0,C 180,E1 -21078.899,E2 -21078.899} C_VEL
LIN {X 0,Y 210.287,Z 689.145,A -85,B 0,C 180,E1 -21081.016,E2 -21081.016} C_VEL
LIN {X 0,Y 211.489,Z 675.1,A -85,B 0,C 180,E1 -21082.725,E2 -21082.725} C_VEL
LIN {X 0,Y 212.687,Z 660.458,A -85,B 0,C 180,E1 -21084.072,E2 -21084.072} C_VEL
LIN {X 0,Y 214.055,Z 638.502,A -85,B 0,C 180,E1 -21085.461,E2 -21085.461} C_VEL
LIN {X 0,Y 217.397,Z 583.043,A -85,B 0,C 180,E1 -21088.664,E2 -21088.664} C_VEL
LIN {X 0,Y 214.509,Z 551.963,A -85,B 0,C 180,E1 -21090.69,E2 -21090.69} C_VEL
LIN {X 0,Y 213.664,Z 541.109,A -85,B 0,C 180,E1 -21091.402,E2 -21091.402} C_VEL
LIN {X 0,Y 212.725,Z 537.632,A -85,B 0,C 180,E1 -21091.723,E2 -21091.723} C_VEL
LIN {X 0,Y 210.49,Z 527.02,A -85,B 0,C 180,E1 -21095.754,E2 -21095.754} C_VEL
LIN {X 0,Y 208.192,Z 516.661,A -85,B 0,C 180,E1 -21099.895,E2 -21099.895} C_VEL
LIN {X 0,Y 206.684,Z 509.862,A -85,B 0,C 180,E1 -21102.755,E2 -21102.755} C_VEL
LIN {X 0,Y 206.626,Z 509.873,A -85,B 0,C 180,E1 -21107.135,E2 -21107.135} C_VEL
LIN {X 0,Y 206.69,Z 509.865,A -85,B 0,C 180,E1 -21111.45,E2 -21111.45} C_VEL
LIN {X 0,Y 206.7,Z 509.858,A -85,B 0,C 180,E1 -21114.689,E2 -21114.689} C_VEL
LIN {X 0,Y 206.725,Z 509.86,A -85,B 0,C 180,E1 -21119.339,E2 -21119.339} C_VEL
LIN {X 0,Y 206.734,Z 509.855,A -85,B 0,C 180,E1 -21123.772,E2 -21123.772} C_VEL
LIN {X 0,Y 206.759,Z 509.854,A -85,B 0,C 180,E1 -21128.043,E2 -21128.043} C_VEL
LIN {X 0,Y 206.875,Z 509.835,A -85,B 0,C 180,E1 -21132.197,E2 -21132.197} C_VEL
LIN {X 0,Y 206.915,Z 509.834,A -85,B 0,C 180,E1 -21136.245,E2 -21136.245} C_VEL
LIN {X 0,Y 207.134,Z 509.804,A -85,B 0,C 180,E1 -21140.232,E2 -21140.232} C_VEL
LIN {X 0,Y 207.19,Z 509.798,A -85,B 0,C 180,E1 -21142.202,E2 -21142.202} C_VEL
LIN {X 0,Y 207.387,Z 509.774,A -85,B 0,C 180,E1 -21148.058,E2 -21148.058} C_VEL
LIN {X 0,Y 207.521,Z 509.756,A -85,B 0,C 180,E1 -21150,E2 -21150} C_VEL
LIN {X 0,Y 207.09,Z 509.813,A -85,B 0,C 180,E1 -21153.892,E2 -21153.892} C_VEL
LIN {X 0,Y 207.19,Z 509.797,A -85,B 0,C 180,E1 -21157.798,E2 -21157.798} C_VEL
LIN {X 0,Y 206.985,Z 509.827,A -85,B 0,C 180,E1 -21161.755,E2 -21161.755} C_VEL
LIN {X 0,Y 206.869,Z 509.838,A -85,B 0,C 180,E1 -21165.771,E2 -21165.771} C_VEL
LIN {X 0,Y 206.801,Z 509.849,A -85,B 0,C 180,E1 -21169.867,E2 -21169.867} C_VEL
LIN {X 0,Y 206.765,Z 509.85,A -85,B 0,C 180,E1 -21174.072,E2 -21174.072} C_VEL
LIN {X 0,Y 206.738,Z 509.856,A -85,B 0,C 180,E1 -21178.42,E2 -21178.42} C_VEL
LIN {X 0,Y 206.707,Z 509.859,A -85,B 0,C 180,E1 -21182.956,E2 -21182.956} C_VEL
LIN {X 0,Y 206.723,Z 509.859,A -85,B 0,C 180,E1 -21185.32,E2 -21185.32} C_VEL
LIN {X 0,Y 206.668,Z 509.863,A -85,B 0,C 180,E1 -21190.25,E2 -21190.25} C_VEL
LIN {X 0,Y 206.636,Z 509.871,A -85,B 0,C 180,E1 -21195.581,E2 -21195.581} C_VEL
LIN {X 0,Y 206.779,Z 509.936,A -85,B 0,C 180,E1 -21200.736,E2 -21200.736} C_VEL
LIN {X 0,Y 210.274,Z 525.17,A -85,B 0,C 180,E1 -21205.068,E2 -21205.068} C_VEL
LIN {X 0,Y 213.845,Z 541.475,A -85,B 0,C 180,E1 -21209.511,E2 -21209.511} C_VEL
LIN {X 0,Y 212.689,Z 551.555,A -85,B 0,C 180,E1 -21211.976,E2 -21211.976} C_VEL
LIN {X 0,Y 214.343,Z 575.595,A -85,B 0,C 180,E1 -21213.446,E2 -21213.446} C_VEL
LIN {X 0,Y 215.273,Z 585.989,A -85,B 0,C 180,E1 -21214.083,E2 -21214.083} C_VEL
LIN {X 0,Y 211.511,Z 661.975,A -85,B 0,C 180,E1 -21218.434,E2 -21218.434} C_VEL
LIN {X 0,Y 210.69,Z 675.741,A -85,B 0,C 180,E1 -21219.527,E2 -21219.527} C_VEL
LIN {X 0,Y 209.708,Z 688.648,A -85,B 0,C 180,E1 -21220.928,E2 -21220.928} C_VEL
LIN {X 0,Y 208.581,Z 700.57,A -85,B 0,C 180,E1 -21222.6,E2 -21222.6} C_VEL
LIN {X 0,Y 207.623,Z 711.678,A -85,B 0,C 180,E1 -21224.54,E2 -21224.54} C_VEL
LIN {X 0,Y 206.783,Z 720.878,A -85,B 0,C 180,E1 -21226.487,E2 -21226.487} C_VEL
LIN {X 0,Y 205.903,Z 731.398,A -85,B 0,C 180,E1 -21229.18,E2 -21229.18} C_VEL
LIN {X 0,Y 205.224,Z 740.624,A -85,B 0,C 180,E1 -21232.127,E2 -21232.127} C_VEL
LIN {X 0,Y 204.832,Z 747.254,A -85,B 0,C 180,E1 -21234.717,E2 -21234.717} C_VEL
LIN {X 0,Y 204.669,Z 754.022,A -85,B 0,C 180,E1 -21238.032,E2 -21238.032} C_VEL
LIN {X 0,Y 204.611,Z 758.688,A -85,B 0,C 180,E1 -21240.984,E2 -21240.984} C_VEL
LIN {X 0,Y 204.733,Z 762.274,A -85,B 0,C 180,E1 -21243.937,E2 -21243.937} C_VEL
LIN {X 0,Y 205.543,Z 765.498,A -85,B 0,C 180,E1 -21247.861,E2 -21247.861} C_VEL
LIN {X 0,Y 207.093,Z 767.201,A -85,B 0,C 180,E1 -21251.749,E2 -21251.749} C_VEL
LIN {X 0,Y 209.728,Z 767.325,A -85,B 0,C 180,E1 -21255.55,E2 -21255.55} C_VEL
LIN {X 0,Y 213.155,Z 765.995,A -85,B 0,C 180,E1 -21259.251,E2 -21259.251} C_VEL
LIN {X 0,Y 215.418,Z 764.755,A -85,B 0,C 180,E1 -21261.031,E2 -21261.031} C_VEL
LIN {X 0,Y 220.538,Z 761.057,A -85,B 0,C 180,E1 -21264.474,E2 -21264.474} C_VEL
LIN {X 0,Y 225.038,Z 757.202,A -85,B 0,C 180,E1 -21266.926,E2 -21266.926} C_VEL
LIN {X 0,Y 230.017,Z 752.342,A -85,B 0,C 180,E1 -21269.266,E2 -21269.266} C_VEL
LIN {X 0,Y 236.375,Z 745.271,A -85,B 0,C 180,E1 -21271.854,E2 -21271.854} C_VEL
LIN {X 0,Y 242.381,Z 737.806,A -85,B 0,C 180,E1 -21273.929,E2 -21273.929} C_VEL
LIN {X 0,Y 249.763,Z 727.254,A -85,B 0,C 180,E1 -21276.222,E2 -21276.222} C_VEL
LIN {X 0,Y 253.326,Z 721.58,A -85,B 0,C 180,E1 -21277.178,E2 -21277.178} C_VEL
LIN {X 0,Y 255.638,Z 717.41,A -85,B 0,C 180,E1 -21277.972,E2 -21277.972} C_VEL
LIN {X 0,Y 261.04,Z 705.629,A -85,B 0,C 180,E1 -21280.687,E2 -21280.687} C_VEL
LIN {X 0,Y 263.111,Z 701.103,A -85,B 0,C 180,E1 -21281.357,E2 -21281.357} C_VEL
LIN {X 0,Y 263.869,Z 699.471,A -85,B 0,C 180,E1 -21281.52,E2 -21281.52} C_VEL
LIN {X 0,Y 269.189,Z 687.365,A -85,B 0,C 180,E1 -21282.497,E2 -21282.497} C_VEL
LIN {X 0,Y 273.821,Z 674.256,A -85,B 0,C 180,E1 -21283.291,E2 -21283.291} C_VEL
LIN {X 0,Y 280.059,Z 651.435,A -85,B 0,C 180,E1 -21284.307,E2 -21284.307} C_VEL
LIN {X 0,Y 273.784,Z 673.727,A -85,B 0,C 180,E1 -21285.355,E2 -21285.355} C_VEL
LIN {X 0,Y 268.764,Z 687.841,A -85,B 0,C 180,E1 -21286.135,E2 -21286.135} C_VEL
LIN {X 0,Y 263.031,Z 700.644,A -85,B 0,C 180,E1 -21287.051,E2 -21287.051} C_VEL
LIN {X 0,Y 256.815,Z 712.61,A -85,B 0,C 180,E1 -21288.202,E2 -21288.202} C_VEL
LIN {X 0,Y 249.065,Z 725.328,A -85,B 0,C 180,E1 -21289.879,E2 -21289.879} C_VEL
LIN {X 0,Y 241.306,Z 736.368,A -85,B 0,C 180,E1 -21291.816,E2 -21291.816} C_VEL
LIN {X 0,Y 233.624,Z 746.118,A -85,B 0,C 180,E1 -21294.083,E2 -21294.083} C_VEL
LIN {X 0,Y 226.492,Z 754.196,A -85,B 0,C 180,E1 -21296.579,E2 -21296.579} C_VEL
LIN {X 0,Y 220.037,Z 760.795,A -85,B 0,C 180,E1 -21299.267,E2 -21299.267} C_VEL
LIN {X 0,Y 213.601,Z 766.656,A -85,B 0,C 180,E1 -21302.572,E2 -21302.572} C_VEL
LIN {X 0,Y 210.722,Z 769.004,A -85,B 0,C 180,E1 -21304.305,E2 -21304.305} C_VEL
LIN {X 0,Y 205.946,Z 772.579,A -85,B 0,C 180,E1 -21307.952,E2 -21307.952} C_VEL
LIN {X 0,Y 202.185,Z 774.714,A -85,B 0,C 180,E1 -21311.769,E2 -21311.769} C_VEL
LIN {X 0,Y 199.548,Z 775.433,A -85,B 0,C 180,E1 -21315.727,E2 -21315.727} C_VEL
LIN {X 0,Y 198.099,Z 774.745,A -85,B 0,C 180,E1 -21319.783,E2 -21319.783} C_VEL
LIN {X 0,Y 197.652,Z 772.584,A -85,B 0,C 180,E1 -21323.877,E2 -21323.877} C_VEL
LIN {X 0,Y 197.754,Z 769.894,A -85,B 0,C 180,E1 -21326.944,E2 -21326.944} C_VEL
LIN {X 0,Y 197.986,Z 767.462,A -85,B 0,C 180,E1 -21329.11,E2 -21329.11} C_VEL
LIN {X 0,Y 197.713,Z 770.589,A -85,B 0,C 180,E1 -21332.037,E2 -21332.037} C_VEL
LIN {X 0,Y 197.576,Z 773.038,A -85,B 0,C 180,E1 -21335.132,E2 -21335.132} C_VEL
LIN {X 0,Y 197.637,Z 774.625,A -85,B 0,C 180,E1 -21338.178,E2 -21338.178} C_VEL
LIN {X 0,Y 198.538,Z 775.668,A -85,B 0,C 180,E1 -21342.263,E2 -21342.263} C_VEL
LIN {X 0,Y 200.482,Z 775.46,A -85,B 0,C 180,E1 -21346.287,E2 -21346.287} C_VEL
LIN {X 0,Y 203.517,Z 774.029,A -85,B 0,C 180,E1 -21350.202,E2 -21350.202} C_VEL
LIN {X 0,Y 207.536,Z 771.408,A -85,B 0,C 180,E1 -21353.977,E2 -21353.977} C_VEL
LIN {X 0,Y 212.575,Z 767.542,A -85,B 0,C 180,E1 -21357.572,E2 -21357.572} C_VEL
LIN {X 0,Y 218.747,Z 762.348,A -85,B 0,C 180,E1 -21360.935,E2 -21360.935} C_VEL
LIN {X 0,Y 225.904,Z 755.71,A -85,B 0,C 180,E1 -21364.055,E2 -21364.055} C_VEL
LIN {X 0,Y 233.868,Z 747.456,A -85,B 0,C 180,E1 -21366.944,E2 -21366.944} C_VEL
LIN {X 0,Y 241.593,Z 738.691,A -85,B 0,C 180,E1 -21369.251,E2 -21369.251} C_VEL
LIN {X 0,Y 249.924,Z 728.238,A -85,B 0,C 180,E1 -21371.364,E2 -21371.364} C_VEL
LIN {X 0,Y 257.456,Z 717.492,A -85,B 0,C 180,E1 -21373.036,E2 -21373.036} C_VEL
LIN {X 0,Y 264.107,Z 707.024,A -85,B 0,C 180,E1 -21374.309,E2 -21374.309} C_VEL
LIN {X 0,Y 271.119,Z 694.351,A -85,B 0,C 180,E1 -21375.467,E2 -21375.467} C_VEL
LIN {X 0,Y 277.591,Z 680.713,A -85,B 0,C 180,E1 -21376.446,E2 -21376.446} C_VEL
LIN {X 0,Y 279.842,Z 675.276,A -85,B 0,C 180,E1 -21376.746,E2 -21376.746} C_VEL
LIN {X 0,Y 280.118,Z 674.443,A -85,B 0,C 180,E1 -21377.079,E2 -21377.079} C_VEL
LIN {X 0,Y 273.488,Z 689.281,A -85,B 0,C 180,E1 -21378.076,E2 -21378.076} C_VEL
LIN {X 0,Y 265.891,Z 703.215,A -85,B 0,C 180,E1 -21379.391,E2 -21379.391} C_VEL
LIN {X 0,Y 258.628,Z 714.732,A -85,B 0,C 180,E1 -21380.817,E2 -21380.817} C_VEL
LIN {X 0,Y 251.145,Z 725.141,A -85,B 0,C 180,E1 -21382.508,E2 -21382.508} C_VEL
LIN {X 0,Y 243.538,Z 734.554,A -85,B 0,C 180,E1 -21384.45,E2 -21384.45} C_VEL
LIN {X 0,Y 237.02,Z 741.838,A -85,B 0,C 180,E1 -21386.377,E2 -21386.377} C_VEL
LIN {X 0,Y 230.091,Z 748.729,A -85,B 0,C 180,E1 -21388.718,E2 -21388.718} C_VEL
LIN {X 0,Y 224.379,Z 753.883,A -85,B 0,C 180,E1 -21390.955,E2 -21390.955} C_VEL
LIN {X 0,Y 217.62,Z 759.229,A -85,B 0,C 180,E1 -21394.152,E2 -21394.152} C_VEL
LIN {X 0,Y 213.183,Z 762.262,A -85,B 0,C 180,E1 -21396.696,E2 -21396.696} C_VEL
LIN {X 0,Y 208.061,Z 765.021,A -85,B 0,C 180,E1 -21400.258,E2 -21400.258} C_VEL
LIN {X 0,Y 203.885,Z 766.36,A -85,B 0,C 180,E1 -21403.992,E2 -21403.992} C_VEL
LIN {X 0,Y 200.947,Z 766.3,A -85,B 0,C 180,E1 -21407.887,E2 -21407.887} C_VEL
LIN {X 0,Y 198.851,Z 764.82,A -85,B 0,C 180,E1 -21411.873,E2 -21411.873} C_VEL
LIN {X 0,Y 197.87,Z 761.839,A -85,B 0,C 180,E1 -21415.926,E2 -21415.926} C_VEL
LIN {X 0,Y 197.582,Z 758.582,A -85,B 0,C 180,E1 -21418.981,E2 -21418.981} C_VEL
LIN {X 0,Y 197.532,Z 754.256,A -85,B 0,C 180,E1 -21422.039,E2 -21422.039} C_VEL
LIN {X 0,Y 197.64,Z 748.351,A -85,B 0,C 180,E1 -21425.331,E2 -21425.331} C_VEL
LIN {X 0,Y 198.102,Z 740.786,A -85,B 0,C 180,E1 -21428.672,E2 -21428.672} C_VEL
LIN {X 0,Y 198.688,Z 732.089,A -85,B 0,C 180,E1 -21431.735,E2 -21431.735} C_VEL
